// TIA Portal project "Esteira_3_V13_SP2_V14_V15" (V15)

(* hardware
DEVICE "S71500/ET200MP station_1"  S7-1500 station
   slot 0: "Rail_0"  6ES7 590-1***0-0AA0
   slot 1: "10D02_PLC"  CPU 1515F-2 PN  6ES7 515-2FM01-0AB0  V1.8
   slot 2: "F-DI 16x24V DC_1"  F-DI 16x24V DC  6ES7 526-1BH00-0AB0  V1.0
      slot 1: "F-DI 16x24V DC_1"  F-DI 16x24V DC  6ES7 526-1BH00-0AB0
   slot 3: "DI 16x24VDC BA_1"  DI 16x24VDC BA  6ES7 521-1BH10-0AA0  V1.0
   slot 4: "DQ 16x24VDC/0.5A BA_1"  DQ 16x24VDC/0.5A BA  6ES7 522-1BH10-0AA0  V1.0
DEVICE "25IHM01"  TP900 Comfort
   slot 0: "HMI"  HMI  6AV2 124-0JC01-0AX0  13.0.1.0
   slot 1: "HMI_RT_1"  TP900 Comfort  6AV2 124-0JC01-0AX0  13.0.1.0
   slot 5: "25IHM01.IE_CP_1"  PROFINET Interface
      slot 1: "PROFINET Interface_1"  PROFINET Interface
         slot 1: "Port_1"  Port
         slot 2: "Port_2"  Port
   slot 7: "25IHM01.MPI/DP_CP_1"  MPI/DP Interface
DEVICE "GSD device_4"  GSD.Device.PN
   slot 0: "Rack"  Rail  V1.0
   slot 0: "21U01_MVK-MPNIO-F"  55556
DEVICE "GSD device_5"  GSD.Device.PN
   slot 0: "Rack"  Rail  V1.0
   slot 0: "20U01_MVK-MPNIO-F"  55556
DEVICE "GSD device_6"  GSD.Device.PN
   slot 0: "Rack"  Rail  V1.0
   slot 0: "09U02_SEW-MDX61B-DFE32B"  182x xxx x  V1.4
      slot 0: "MDX61B+DFE32B V1.4"  182x xxx x  V1.4
DEVICE "SCALANCE X005"  SCALANCE X-Station
   slot 0: "SCALANCE X rack"  Rail
   slot 0: "Switch_1"  6GK5 005-0BA00-1AB2  V1.0
DEVICE "SCALANCE X005_1"  SCALANCE X-Station
   slot 0: "SCALANCE X rack"  Rail
   slot 0: "Switch_2"  6GK5 005-0BA00-1AB2  V1.0
DEVICE "GSD device_1"  GSD.Device.PN
   slot 0: "Rack"  Rail  V1.0
   slot 0: "19U02_Cube67-BN-PNIO"  56526  2
   slot 5: "21U05_56601 DIO16 E 8xM12_2"  56601
   slot 7: "20U05_56601 DIO16 E 8xM12_1"  56601
*)

// ===== PLC "10D02_PLC"  CPU 1515F-2 PN =====
// protected blocks, not shown: "Main_Safety_RTG1", "Main_Safety_RTG1_DB"

VAR_GLOBAL   // PLC tag table "Default tag table"
   "M_Estacao1_Andon" AT %M50.0 : Bool;
   "System_Byte" AT %MB1 : Byte;
   "FirstScan" AT %M1.0 : Bool;
   "DiagStatusUpdate" AT %M1.1 : Bool;
   "AlwaysTRUE" AT %M1.2 : Bool;
   "AlwaysFALSE" AT %M1.3 : Bool;
   "Clock_Byte" AT %MB0 : Byte;
   "Clock_10Hz" AT %M0.0 : Bool;
   "Clock_5Hz" AT %M0.1 : Bool;
   "Clock_2.5Hz" AT %M0.2 : Bool;
   "Clock_2Hz" AT %M0.3 : Bool;
   "Clock_1.25Hz" AT %M0.4 : Bool;
   "Clock_1Hz" AT %M0.5 : Bool;
   "Clock_0.625Hz" AT %M0.6 : Bool;
   "Clock_0.5Hz" AT %M0.7 : Bool;
   "Sempre_0" AT %M2.0 : Bool;
   "IHM_Tempo_Takt" AT %MD4 : Time;
   "IHM_Contagem_Tempo" AT %MD8 : Time;
   "11ME01_Emergência¶Painel Principal" AT %I0.0 : Bool;
   "11ME01_Reserva" AT %I0.1 : Bool;
   "11ME01_Reserva(1)" AT %I0.2 : Bool;
   "11ME01_Reserva(2)" AT %I0.3 : Bool;
   "11ME01_Reserva(3)" AT %I0.4 : Bool;
   "11ME01_Reserva(4)" AT %I0.5 : Bool;
   "11ME01_Reserva(5)" AT %I0.6 : Bool;
   "11ME01_Reserva(6)" AT %I0.7 : Bool;
   "11ME01_Emergência¶Painel Principal(1)" AT %I1.0 : Bool;
   "11ME01_Reserva(7)" AT %I1.1 : Bool;
   "11ME01_Reserva(8)" AT %I1.2 : Bool;
   "11ME01_Reset" AT %I1.3 : Bool;
   "11ME01_Reserva(9)" AT %I1.4 : Bool;
   "11ME01_Reserva(10)" AT %I1.5 : Bool;
   "11ME01_Reserva(11)" AT %I1.6 : Bool;
   "11ME01_Reserva(12)" AT %I1.7 : Bool;
   "12ME02_Termostato¶Painel" AT %I12.0 : Bool;
   "12ME02_Disjuntor¶Serviço Ok" AT %I12.1 : Bool;
   "12ME02_Disjuntor¶Tomada Ok" AT %I12.2 : Bool;
   "12ME02_Disjuntor¶Iluminação Ok" AT %I12.3 : Bool;
   "12ME02_Disjuntor¶Ar Condicionado Ok" AT %I12.4 : Bool;
   "12ME02_Disjuntor¶08F03 Ok" AT %I12.5 : Bool;
   "12ME02_Disjuntor¶Freio Ok" AT %I12.6 : Bool;
   "12ME02_Disjuntor¶Drive Ok" AT %I12.7 : Bool;
   "12ME02_Aquecimento¶Resistor Frenagem" AT %I13.0 : Bool;
   "12ME02_Disjuntor¶Ventilação Ok" AT %I13.1 : Bool;
   "12ME02_Reset_Emergencia" AT %I13.2 : Bool;
   "12ME02_Reserva(1)" AT %I13.3 : Bool;
   "12ME02_Reserva(2)" AT %I13.4 : Bool;
   "12ME02_Reserva(3)" AT %I13.5 : Bool;
   "12ME02_Reserva(4)" AT %I13.6 : Bool;
   "12ME02_Reserva(5)" AT %I13.7 : Bool;
   "15MS02_Reserva" AT %Q5.0 : Bool;
   "15MS02_Sirene_Giro" AT %Q5.1 : Bool;
   "15MS02_Reserva(2)" AT %Q5.2 : Bool;
   "15MS02_Reset" AT %Q5.3 : Bool;
   "15MS02_Torre de Sinalização¶Azul" AT %Q5.4 : Bool;
   "15MS02_Torre de Sinalização¶Verde" AT %Q5.5 : Bool;
   "15MS02_Torre de Sinalização¶Amarela" AT %Q5.6 : Bool;
   "15MS02_Torre de Sinalização¶Vermelha" AT %Q5.7 : Bool;
   "15MS02_Liga Ventilação¶Forçada" AT %Q6.0 : Bool;
   "15MS02_Reset_Rele_Emergencia" AT %Q6.1 : Bool;
   "15MS02_Reserva(4)" AT %Q6.2 : Bool;
   "15MS02_Reserva(5)" AT %Q6.3 : Bool;
   "15MS02_Reserva(6)" AT %Q6.4 : Bool;
   "15MS02_Reserva(7)" AT %Q6.5 : Bool;
   "15MS02_Reserva(8)" AT %Q6.6 : Bool;
   "15MS02_Reserva(9)" AT %Q6.7 : Bool;
   "20U1_Ack_Necessario" AT %I25.0 : Bool;
   "21U1_Ack_Necessario" AT %I34.0 : Bool;
   "22U1_Ack_Necessario" AT %I37.0 : Bool;
   "23U1_Ack_Necessario" AT %I68.0 : Bool;
   "20U1_GRUPO_OK" AT %I25.1 : Bool;
   "21U1_GRUPO_OK" AT %I34.1 : Bool;
   "22U1_GRUPO_OK" AT %I37.1 : Bool;
   "23U1_GRUPO_OK" AT %I68.1 : Bool;
   "IHM_Alarmes_Teste" AT %MB3 : Byte;
   "Contador_Cabinas" AT %MW12 : Int;
   "Ciclo_Giro" AT %MW14 : Word;
   "TESTES_MANUAIS" AT %M2.3 : Bool;
   "TESTE_LAMPADAS" AT %M20.0 : Bool;
END_VAR

VAR_GLOBAL   // PLC tag table "20U05"
   "20U05_Libera¶Estação 10" AT %I140.0 : Bool;
   "20U05_Reserva" AT %Q140.1 : Bool;
   "20U05_Libera¶Estação 20" AT %I140.2 : Bool;
   "20U05_Reserva(1)" AT %Q140.3 : Bool;
   "20U05_Reserva(2)" AT %I140.4 : Bool;
   "20U05_Reserva(3)" AT %Q140.5 : Bool;
   "20U05_Reserva(4)" AT %I140.6 : Bool;
   "20U05_Reserva(5)" AT %Q140.7 : Bool;
   "20U05_Apoio¶Estação 10" AT %I141.0 : Bool;
   "20U05_Reserva(6)" AT %Q141.1 : Bool;
   "20U05_Apoio¶Estação 20" AT %I141.2 : Bool;
   "20U05_Reserva(7)" AT %Q141.3 : Bool;
   "20U05_Reserva(8)" AT %I141.4 : Bool;
   "20U05_Reserva(9)" AT %Q141.5 : Bool;
   "20U05_Reserva(10)" AT %I141.6 : Bool;
   "20U05_Reserva(11)" AT %Q141.7 : Bool;
END_VAR

VAR_GLOBAL   // PLC tag table "20U01"
   "20U01_Reserva" AT %I116.0 : Bool;
   "20U01_Reserva(1)" AT %I116.1 : Bool;
   "20U01_Reserva(2)" AT %I116.2 : Bool;
   "20U01_Emergência¶Estação 1" AT %I116.3 : Bool;
   "20U01_Reserva(3)" AT %I116.4 : Bool;
   "20U01_Reserva(4)" AT %I116.5 : Bool;
   "20U01_Reserva(5)" AT %I116.6 : Bool;
   "20U01_Reserva(6)" AT %I116.7 : Bool;
   "20U01_Emergência¶Estação 2" AT %I117.0 : Bool;
   "20U01_Reserva(7)" AT %I117.1 : Bool;
   "20U01_Reserva(8)" AT %I117.2 : Bool;
   "20U01_Reserva(9)" AT %I117.3 : Bool;
   "20U01_Reserva(10)" AT %I117.4 : Bool;
   "20U01_Reserva(11)" AT %I117.5 : Bool;
   "20U01_Reserva(12)" AT %I117.6 : Bool;
   "20U01_Reserva(13)" AT %I117.7 : Bool;
   "20U1_Reseta_Modulo" AT %Q7.0 : Bool;
   "Muting_Cortina" AT %M2.1 : Bool;
   "Emergencia_Cortina" AT %M2.2 : Bool;
END_VAR

VAR_GLOBAL   // PLC tag table "21U01"
   "21U01_Cortina_Saida" AT %I122.0 : Bool;
   "21U01_Reserva(1)" AT %I122.1 : Bool;
   "21U01_Reserva(2)" AT %I122.2 : Bool;
   "21U01_Emergência¶Estação 3" AT %I122.3 : Bool;
   "21U01_Reserva(3)" AT %I122.4 : Bool;
   "21U01_Reserva(4)" AT %I122.5 : Bool;
   "21U01_Reserva(5)" AT %I122.6 : Bool;
   "21U01_Reserva(6)" AT %I122.7 : Bool;
   "21U01_Emergência¶Estação 4" AT %I123.0 : Bool;
   "21U01_Reserva(7)" AT %I123.1 : Bool;
   "21U01_Reserva(8)" AT %I123.2 : Bool;
   "21U01_Reserva(9)" AT %I123.3 : Bool;
   "21U01_Reserva(10)" AT %I123.4 : Bool;
   "21U01_Reserva(11)" AT %I123.5 : Bool;
   "21U01_Reserva(12)" AT %I123.6 : Bool;
   "21U01_Reserva(13)" AT %I123.7 : Bool;
   "21U1_Reseta_Modulo" AT %Q8.0 : Bool;
END_VAR

VAR_GLOBAL   // PLC tag table "21U05"
   "21U05_Libera¶Estação 30" AT %I144.0 : Bool;
   "21U05_Reserva" AT %Q144.1 : Bool;
   "21U05_Libera¶Estação 40" AT %I144.2 : Bool;
   "21U05_Reserva(1)" AT %Q144.3 : Bool;
   "21U05_Cabine_Retirada" AT %I144.4 : Bool;
   "21U05_Reserva(3)" AT %Q144.5 : Bool;
   "21U05_Reserva(4)" AT %I144.6 : Bool;
   "21U05_Reserva(5)" AT %Q144.7 : Bool;
   "21U05_Apoio¶Estação 30" AT %I145.0 : Bool;
   "21U05_Reserva(6)" AT %Q145.1 : Bool;
   "21U05_Apoio¶Estação 40" AT %I145.2 : Bool;
   "21U05_Reserva(7)" AT %Q145.3 : Bool;
   "21U05_Reserva(8)" AT %I145.4 : Bool;
   "21U05_Reserva(9)" AT %Q145.5 : Bool;
   "21U05_Reserva(10)" AT %I145.6 : Bool;
   "21U05_Reserva(11)" AT %Q145.7 : Bool;
END_VAR

DATA_BLOCK "ANDON_DB"   // DB2
{ S7_Optimized_Access := 'TRUE' }
VERSION : 0.1
// stored: InstanceOfName ANDON
"ANDON"
BEGIN
END_DATA_BLOCK

DATA_BLOCK "Multiplo_Uso_DB"   // DB5
{ S7_Optimized_Access := 'TRUE' }
VERSION : 0.1
   VAR
      HORA_Atual : Time_Of_Day;
      DATA_Atual : DTL;
   END_VAR
   VAR RETAIN
      T_Takt : IEC_COUNTER;
   END_VAR
   VAR
      retorno_Data : Int;
   END_VAR
   VAR RETAIN
      INICIO_JORNADA : DTL;
      FINAL_JORNADA : DTL;
      INICIO_ALMOÇO : DTL;
   END_VAR
   VAR
      FINAL_ALMOÇO : DTL;
      EM_JORNADA : Bool;
      EM_JORNADA_CMP : Bool;
   END_VAR
   VAR RETAIN
      IHM_TAKT_MINUTOS : Int;
      IHM_TAKT_SEGUNDOS : Int;
      TAKT_SEGUNDOS : Int;
   END_VAR
   VAR
      FINAL_DO_TAKT : Bool;
      Contagem_Takt : Int;
      Emergencia_Principal_OK : Bool;
      Emergencia_OP10_OK : Bool;
      Emergencia_OP20_OK : Bool;
      Emergencia_OP30_OK : Bool;
      Emergencia_OP40_OK : Bool;
      Emergencia_OP50_OK : Bool;
      Emergencia_OP60_OK : Bool;
      Emergencia_OP70_OK : Bool;
      Emergencia_OP80_OK : Bool;
      EMERGENCIAS_OK : Bool;
      OPERACAO10_OK : Bool;
      OPERACAO20_OK : Bool;
      OPERACAO30_OK : Bool;
      OPERACAO40_OK : Bool;
      OPERACAO50_OK : Bool;
      OPERACAO60_OK : Bool;
      OPERACAO70_OK : Bool;
      OPERACAO80_OK : Bool;
      OPERACOES_OK : Bool;
      Roda_Linha : Bool;
      Roda_Linha_cmp : Bool;
   END_VAR
   VAR RETAIN
      CONTAGEM_CABINAS : Int;
      TOTAL_CABINAS_TURNO : Int;
   END_VAR
   VAR
      GMT_Brasilia : Time := T#3h;
      Fim_De_Producao : Bool;
      Fim_De_Producao_cmp : Bool;
   END_VAR
   VAR RETAIN
      DESABILITA_OP10 : Bool;
      DESABILITA_OP20 : Bool;
      DESABILITA_OP30 : Bool;
      DESABILITA_OP40 : Bool;
      DESABILITA_OP50 : Bool;
      DESABILITA_OP60 : Bool;
      DESABILITA_OP70 : Bool;
      DESABILITA_OP80 : Bool;
      IHM_Velocidade_Automatico : Int := 10;
      IHM_Velocidade_Manual : Int := 4;
      IHM_Descolamento_Cabinas_mm : DInt := 5825;
   END_VAR
   VAR
      IHM_Modo_Manual : Bool;
      IHM_Modo_Manual_cmp : Bool;
      IHM_Modo_Automatico : Bool;
      IHM_Modo_Automatico_cmp : Bool;
      IHM_Jog_CW : Bool;
      IHM_Jog_CCW : Bool;
      IHM_Posicao_Atual : DInt;
      IHM_Velocidade_Atual : Int;
      T_RESET_RELE_SEG : IEC_TIMER;
      IHM_HABILITA_DRIVER : Bool;
      IHM_HABILITA_DRIVER_CMP : Bool;
      ZERA_POSICAO : Bool;
      RESETA_TAKT : Bool;
      PARAR_OP10 : Bool;
      PARAR_OP20 : Bool;
      PARAR_OP30 : Bool;
      PARAR_OP40 : Bool;
      PARAR_OP50 : Bool;
      PARAR_OP60 : Bool;
      PARAR_OP70 : Bool;
      PARAR_OP80 : Bool;
      Ciclo_Giro : Int;
      Shifter_Giro : Bool;
      T_Reset_Takt : IEC_TIMER;
      T_Retirada_Cabine : IEC_TIMER;
      CABINE_RETIRADA : Bool;
      Emergencia_Cortina_Saida_OK : Bool;
      Muting_Cortina : Bool;
      T_SIRENE : IEC_TIMER;
      Sirene_Giro : Bool;
      Tempo_Sirene : Time;
   END_VAR
   VAR RETAIN
      IHM_Tempo_Aviso1 : Int;
      IHM_Tempo_Aviso2 : Int;
   END_VAR
   VAR
      Inicio_Aviso1 : Int;
      Final_Aviso1 : Int;
      Inicio_Aviso2 : Int;
      Final_Aviso2 : Int;
      IHM_Zerar_Contagem : Bool;
      IHM_Zerar_Posicao_Esteira : Bool;
      IHM_Zerar_Takt : Bool;
      Tempo_OP10 : Int;
      Tempo_OP20 : Int;
      Tempo_OP30 : Int;
      Tempo_OP40 : Int;
      Stop_Time_OP10 : Int;
      Stop_Time_OP20 : Int;
      Stop_Time_OP30 : Int;
      Stop_Time_OP40 : Int;
   END_VAR
BEGIN
END_DATA_BLOCK

DATA_BLOCK "ALARMES_DB"   // DB12
{ S7_Optimized_Access := 'FALSE' }
VERSION : 0.1
   VAR
      DBW0 : Int;
      DBW1 : Int;
      DBW2 : Int;
      DBW3 : Int;
   END_VAR
BEGIN
END_DATA_BLOCK

DATA_BLOCK "DB_Global_Sistema"   // DB23
{ S7_Optimized_Access := 'FALSE' }
VERSION : 0.1
   VAR
      TEMPO_TAKT : Int;
      Apoio_OP10 : Bool;
      Apoio_OP20 : Bool;
      Apoio_OP30 : Bool;
      Apoio_OP40 : Bool;
      Apoio_OP50 : Bool;
      Apoio_OP60 : Bool;
      Apoio_OP70 : Bool;
      Apoio_OP80 : Bool;
      Contagem_Cabinas : Int;
      Stop_Time : Int;
      Cabinas_Programadas : Int;
   END_VAR
BEGIN
END_DATA_BLOCK

DATA_BLOCK "Modulo_259"   // DB286
{ S7_Optimized_Access := 'TRUE' }
VERSION : 0.1
   VAR
      IO_ADDRESS_or_HW_IDENTIFIER : Hw_Io := 318;   // S71xxxx: assign HW_Identifier; S74xx/3xx assign Peripheral address
      INHIBIT : Bool;   // false: Contr. inhibit; true: enable
      ENABLE_RAPID_STOP : Bool;   // false: rapid stop; true: enable
      ENABLE : Bool;   // false: stop; true: enable
      RESET : Bool;
      Start : Bool;
      JOG_PLUS_MODE : Bool;   // select Jog+_Mode
      JOG_MINUS_MODE : Bool;   // select Jog-_Mode
      REF_TRAVEL_MODE : Bool;   // select Reference_Travel_Mode
      AUTO_OPT : Bool;   // select AUTO_OPT_Mode
      AUTO_CW : Bool;   // select AUTO_CW_Mode
      AUTO_CCW : Bool;   // select AUTO_CCW_Mode
      AUTO_PULS_CW : Bool;   // select AUTO_PULS_CW_Mode
      AUTO_PULS_CCW : Bool;   // select AUTO_PULS_CCW_Mode
      SETPOINT_POS : DInt := 0;
      SETPOINT_SPEED : Int := 4;
      START_RAMP : Int := 1001;   // Attention: Avoid Ramp = 0!
      STOP_RAMP : Int := 2002;   // Attention: Avoid Ramp = 0!
      COMMUNICATION_OK : Bool;   // DPRD_DAT & DPWR_DAT: Return Value = 0 / SFC14/SFC15: Return Value = 0
      FAULT_OF_AXIS : Bool;   // A fault is active, if the inverter is not ready for operation AND the error bit has been set.
      WARNING_OF_AXIS : Bool;   // A warning is active, if the inverter is still ready for operation AND the error bit has been set.
      INVERTER_READY : Bool;
      REFERENCED : Bool;
      TARGET_POS_REACHED : Bool;
      AXIS_INTERLOCKED : Bool;   // mode selection is illogical (no mode or several modes selected) / die Modeanwahl ist unplausibel (kein Mode oder mehrere Modi angewählt)
      FAULT_NO : Int;
      ACTUAL_POSITION : DInt;
      ACTUAL_SPEED : Int;
      ACTUAL_CURRENT : Int;
   END_VAR
BEGIN
END_DATA_BLOCK

// folder: BANCO

DATA_BLOCK "Banco_Hora_Operacoes"   // DB13
{ S7_Optimized_Access := 'FALSE' }
VERSION : 0.1
   VAR
      Produto_1 : Struct
         Data_e_Hora : DTL;
         Tempo_OP10 : Int;
         Tempo_OP20 : Int;
         Tempo_OP30 : Int;
         Tempo_OP40 : Int;
         Tempo_OP50 : Int;
         Tempo_OP60 : Int;
         Tempo_OP70 : Int;
         Tempo_OP80 : Int;
         Stop_Time_OP10 : Int;
         Stop_Time_OP20 : Int;
         Stop_Time_OP30 : Int;
         Stop_Time_OP40 : Int;
         Stop_Time_OP50 : Int;
         Stop_Time_OP60 : Int;
         Stop_Time_OP70 : Int;
         Stop_Time_OP80 : Int;
      END_STRUCT;
   END_VAR
BEGIN
END_DATA_BLOCK

// folder: DB_OPERACOES

DATA_BLOCK "Operacao_20_DB"   // DB3
{ S7_Optimized_Access := 'TRUE' }
VERSION : 0.1
// stored: InstanceOfName Operacao
"Operacao"
BEGIN
END_DATA_BLOCK

DATA_BLOCK "Operacao_10_DB"   // DB4
{ S7_Optimized_Access := 'TRUE' }
VERSION : 0.1
// stored: InstanceOfName Operacao
"Operacao"
BEGIN
END_DATA_BLOCK

DATA_BLOCK "Operacao_30_DB"   // DB6
{ S7_Optimized_Access := 'TRUE' }
VERSION : 0.1
// stored: InstanceOfName Operacao
"Operacao"
BEGIN
END_DATA_BLOCK

DATA_BLOCK "Operacao_40_DB"   // DB7
{ S7_Optimized_Access := 'TRUE' }
VERSION : 0.1
// stored: InstanceOfName Operacao
"Operacao"
BEGIN
END_DATA_BLOCK

DATA_BLOCK "Operacao_50_DB"   // DB8
{ S7_Optimized_Access := 'TRUE' }
VERSION : 0.1
// stored: InstanceOfName Operacao
"Operacao"
BEGIN
END_DATA_BLOCK

DATA_BLOCK "Operacao_60_DB"   // DB9
{ S7_Optimized_Access := 'TRUE' }
VERSION : 0.1
// stored: InstanceOfName Operacao
"Operacao"
BEGIN
END_DATA_BLOCK

DATA_BLOCK "Operacao_70_DB"   // DB10
{ S7_Optimized_Access := 'TRUE' }
VERSION : 0.1
// stored: InstanceOfName Operacao
"Operacao"
BEGIN
END_DATA_BLOCK

DATA_BLOCK "Operacao_80_DB"   // DB11
{ S7_Optimized_Access := 'TRUE' }
VERSION : 0.1
// stored: InstanceOfName Operacao
"Operacao"
BEGIN
END_DATA_BLOCK

// folder: (top level)

FUNCTION_BLOCK "Operacao"   // FB2, LAD
{ S7_Optimized_Access := 'TRUE' }
VERSION : 0.1
   VAR_INPUT
      Parar_Linha : Bool;
      Emergencia_OK : Bool;
      Emergencia_OP_OK : Bool;
   END_VAR
   VAR_OUTPUT
      Operacao_OK : Bool;
      Tempo_Da_Operacao : Int;
      Stop_Time : Int;
   END_VAR
   VAR
      Operacao_OK_cmp : Bool;
   END_VAR
   VAR_TEMP   // added for the SCL form of the ladder/FBD networks
      _w1 : Bool;
   END_VAR
BEGIN

REGION Network 1: operacao ok
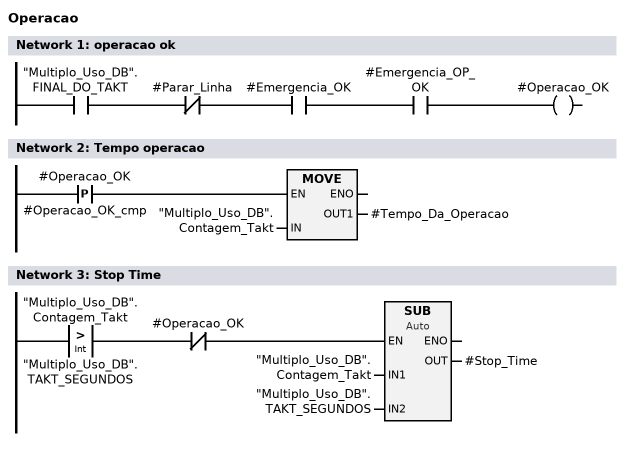
   RUNG wire#powerrail
      Contact( "Multiplo_Uso_DB".FINAL_DO_TAKT )
      I_Contact( #Parar_Linha )
      Contact( #Emergencia_OK )
      Contact( #Emergencia_OP_OK )
      Coil( #Operacao_OK )
   END_RUNG
   // the same network as SCL:
   #Operacao_OK := "Multiplo_Uso_DB".FINAL_DO_TAKT AND NOT #Parar_Linha AND #Emergencia_OK AND #Emergencia_OP_OK;
END_REGION

REGION Network 2: Tempo operacao
   RUNG wire#powerrail
      P_Contact(operand := #Operacao_OK, bit := #Operacao_OK_cmp)
      Move(in := "Multiplo_Uso_DB".Contagem_Takt, out1 => #Tempo_Da_Operacao)
   END_RUNG
   // the same network as SCL:
   #_w1 := #Operacao_OK AND NOT #Operacao_OK_cmp;   // rising edge of #Operacao_OK
   #Operacao_OK_cmp := #Operacao_OK;
   IF #_w1 THEN #Tempo_Da_Operacao := "Multiplo_Uso_DB".Contagem_Takt; END_IF;
END_REGION

REGION Network 3: Stop Time
   RUNG wire#powerrail
      { S7_Templates := "SrcType := Int" } GT_Contact(in1 := "Multiplo_Uso_DB".Contagem_Takt, in2 := "Multiplo_Uso_DB".TAKT_SEGUNDOS)
      I_Contact( #Operacao_OK )
      Sub(in1 := "Multiplo_Uso_DB".Contagem_Takt, in2 := "Multiplo_Uso_DB".TAKT_SEGUNDOS, out => #Stop_Time)
   END_RUNG
   // the same network as SCL:
   IF ("Multiplo_Uso_DB".Contagem_Takt > "Multiplo_Uso_DB".TAKT_SEGUNDOS) AND NOT #Operacao_OK THEN
       #Stop_Time := "Multiplo_Uso_DB".Contagem_Takt - "Multiplo_Uso_DB".TAKT_SEGUNDOS;
   END_IF;
END_REGION
END_FUNCTION_BLOCK

FUNCTION_BLOCK "ANDON"   // FB3, LAD
{ S7_Optimized_Access := 'TRUE' }
VERSION : 0.1
   VAR_INPUT
      FINAL_JORNADA : DTL;
      INICIO_JORNADA : DTL;
      INICIO_ALMOÇO : DTL;
   END_VAR
   VAR_OUTPUT
      EM_JORNADA : Bool;
      FINAL_DE_TAKT : Bool;
   END_VAR
   VAR
      FINAL_ALMOÇO : DTL;
      INICIAR_CONTAGEM : Bool;
      INICIAR_CONTAGEM_cmp : Bool;
      MINUTOS_P_SEGUNDOS : Int;
      T_SIRENE_INT : Int;
   END_VAR
BEGIN

REGION Network 1
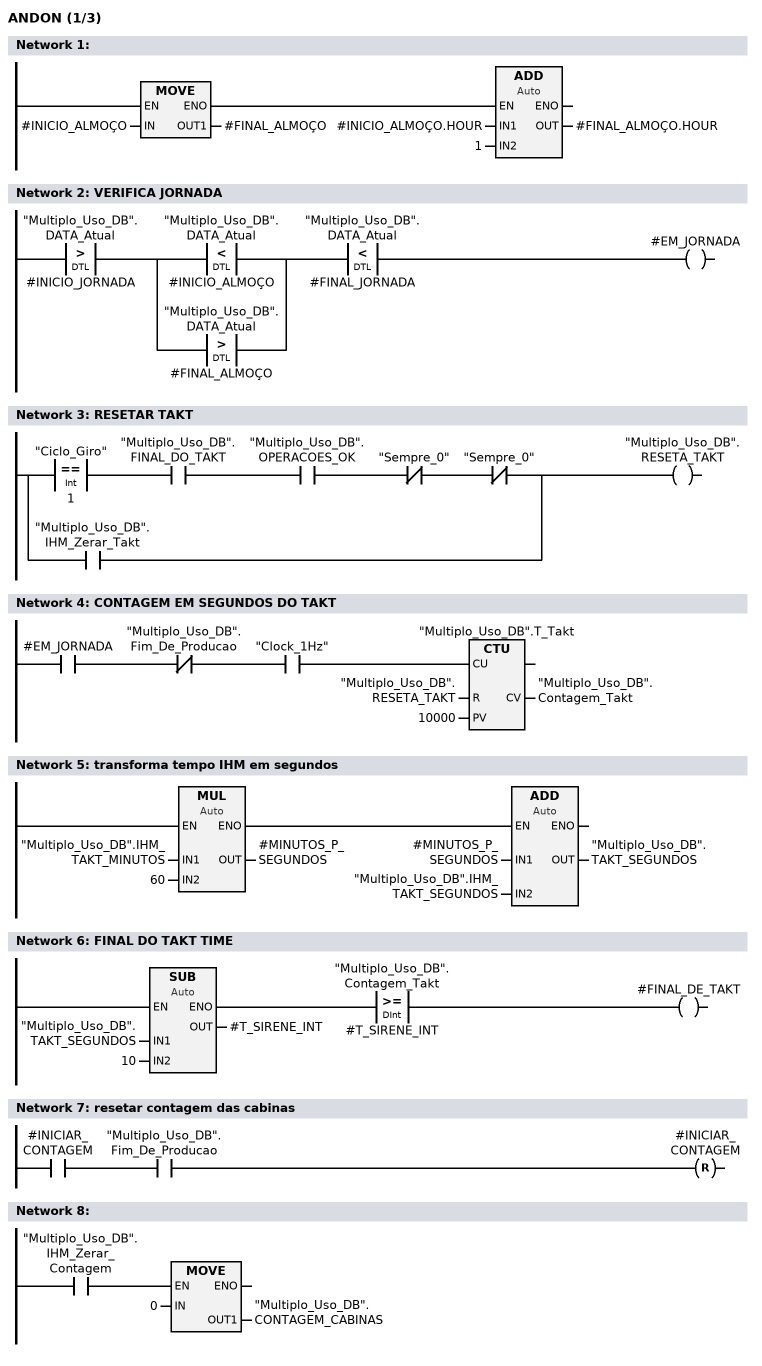
   RUNG wire#powerrail
      Move(in := #INICIO_ALMOÇO, out1 => #FINAL_ALMOÇO)
      Add(in1 := #INICIO_ALMOÇO.HOUR, in2 := 1, out => #FINAL_ALMOÇO.HOUR)
   END_RUNG
   // the same network as SCL:
   #FINAL_ALMOÇO := #INICIO_ALMOÇO;
   #FINAL_ALMOÇO.HOUR := #INICIO_ALMOÇO.HOUR + 1;
END_REGION

REGION Network 2: VERIFICA JORNADA
   RUNG wire#powerrail
      { S7_Templates := "SrcType := DTL" } GT_Contact(in1 := "Multiplo_Uso_DB".DATA_Atual, in2 := #INICIO_JORNADA)
      wire#w1
      { S7_Templates := "SrcType := DTL" } LT_Contact(in1 := "Multiplo_Uso_DB".DATA_Atual, in2 := #INICIO_ALMOÇO)
      wire#w2
      { S7_Templates := "SrcType := DTL" } LT_Contact(in1 := "Multiplo_Uso_DB".DATA_Atual, in2 := #FINAL_JORNADA)
      Coil( #EM_JORNADA )
   END_RUNG
   RUNG wire#w1
      { S7_Templates := "SrcType := DTL" } GT_Contact(in1 := "Multiplo_Uso_DB".DATA_Atual, in2 := #FINAL_ALMOÇO)
   END_RUNG wire#w2
   // the same network as SCL:
   #EM_JORNADA := ("Multiplo_Uso_DB".DATA_Atual > #INICIO_JORNADA) AND (("Multiplo_Uso_DB".DATA_Atual < #INICIO_ALMOÇO) OR ("Multiplo_Uso_DB".DATA_Atual > #FINAL_ALMOÇO)) AND ("Multiplo_Uso_DB".DATA_Atual < #FINAL_JORNADA);
END_REGION

REGION Network 3: RESETAR TAKT
   RUNG wire#powerrail
      { S7_Templates := "SrcType := Int" } EQ_Contact(in1 := "Ciclo_Giro", in2 := 1)
      Contact( "Multiplo_Uso_DB".FINAL_DO_TAKT )
      Contact( "Multiplo_Uso_DB".OPERACOES_OK )
      I_Contact( "Sempre_0" )
      I_Contact( "Sempre_0" )
      wire#w1
      Coil( "Multiplo_Uso_DB".RESETA_TAKT )
   END_RUNG
   RUNG wire#powerrail
      Contact( "Multiplo_Uso_DB".IHM_Zerar_Takt )
   END_RUNG wire#w1
   // the same network as SCL:
   "Multiplo_Uso_DB".RESETA_TAKT := (("Ciclo_Giro" = 1) AND "Multiplo_Uso_DB".FINAL_DO_TAKT AND "Multiplo_Uso_DB".OPERACOES_OK AND NOT "Sempre_0" AND NOT "Sempre_0") OR "Multiplo_Uso_DB".IHM_Zerar_Takt;
END_REGION

REGION Network 4: CONTAGEM EM SEGUNDOS DO TAKT
   "Multiplo_Uso_DB".T_Takt.CTU(CU := #EM_JORNADA AND NOT "Multiplo_Uso_DB".Fim_De_Producao AND "Clock_1Hz",
                           R := "Multiplo_Uso_DB".RESETA_TAKT,
                           PV := 10000,
                           CV => "Multiplo_Uso_DB".Contagem_Takt);
END_REGION

REGION Network 5: transforma tempo IHM em segundos
   RUNG wire#powerrail
      Mul(in1 := "Multiplo_Uso_DB".IHM_TAKT_MINUTOS, in2 := 60, out => #MINUTOS_P_SEGUNDOS)
      Add(in1 := #MINUTOS_P_SEGUNDOS, in2 := "Multiplo_Uso_DB".IHM_TAKT_SEGUNDOS, out => "Multiplo_Uso_DB".TAKT_SEGUNDOS)
   END_RUNG
   // the same network as SCL:
   #MINUTOS_P_SEGUNDOS := "Multiplo_Uso_DB".IHM_TAKT_MINUTOS * 60;
   "Multiplo_Uso_DB".TAKT_SEGUNDOS := #MINUTOS_P_SEGUNDOS + "Multiplo_Uso_DB".IHM_TAKT_SEGUNDOS;
END_REGION

REGION Network 6: FINAL DO TAKT TIME
   RUNG wire#powerrail
      Sub(in1 := "Multiplo_Uso_DB".TAKT_SEGUNDOS, in2 := 10, out => #T_SIRENE_INT)
      { S7_Templates := "SrcType := DInt" } GE_Contact(in1 := "Multiplo_Uso_DB".Contagem_Takt, in2 := #T_SIRENE_INT)
      Coil( #FINAL_DE_TAKT )
   END_RUNG
   // the same network as SCL:
   #T_SIRENE_INT := "Multiplo_Uso_DB".TAKT_SEGUNDOS - 10;
   #FINAL_DE_TAKT := "Multiplo_Uso_DB".Contagem_Takt >= #T_SIRENE_INT;
END_REGION

REGION Network 7: resetar contagem das cabinas
   RUNG wire#powerrail
      Contact( #INICIAR_CONTAGEM )
      Contact( "Multiplo_Uso_DB".Fim_De_Producao )
      R_Coil( #INICIAR_CONTAGEM )
   END_RUNG
   // the same network as SCL:
   IF #INICIAR_CONTAGEM AND "Multiplo_Uso_DB".Fim_De_Producao THEN #INICIAR_CONTAGEM := FALSE; END_IF;
END_REGION

REGION Network 8
   RUNG wire#powerrail
      Contact( "Multiplo_Uso_DB".IHM_Zerar_Contagem )
      Move(in := 0, out1 => "Multiplo_Uso_DB".CONTAGEM_CABINAS)
   END_RUNG
   // the same network as SCL:
   IF "Multiplo_Uso_DB".IHM_Zerar_Contagem THEN "Multiplo_Uso_DB".CONTAGEM_CABINAS := 0; END_IF;
END_REGION

REGION Network 9: Sinaliza fim de produção
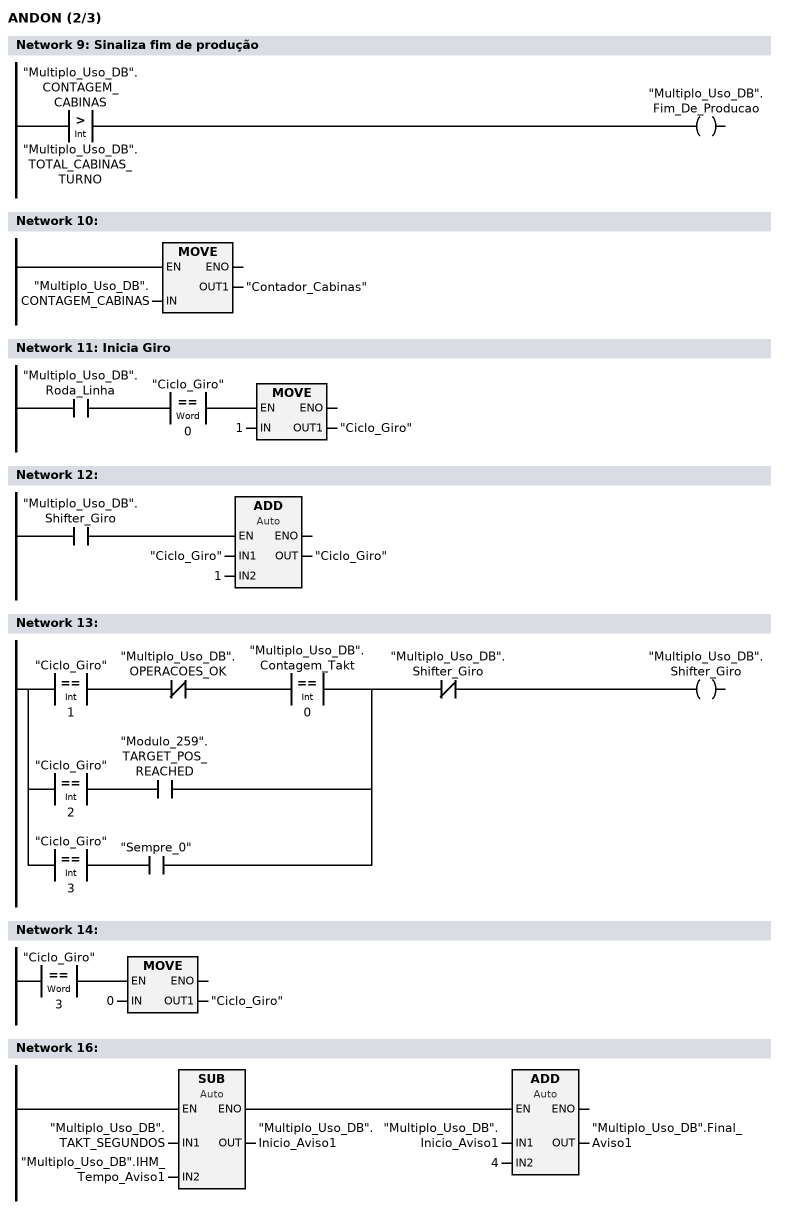
   RUNG wire#powerrail
      { S7_Templates := "SrcType := Int" } GT_Contact(in1 := "Multiplo_Uso_DB".CONTAGEM_CABINAS, in2 := "Multiplo_Uso_DB".TOTAL_CABINAS_TURNO)
      Coil( "Multiplo_Uso_DB".Fim_De_Producao )
   END_RUNG
   // the same network as SCL:
   "Multiplo_Uso_DB".Fim_De_Producao := "Multiplo_Uso_DB".CONTAGEM_CABINAS > "Multiplo_Uso_DB".TOTAL_CABINAS_TURNO;
END_REGION

REGION Network 10
   RUNG wire#powerrail
      Move(in := "Multiplo_Uso_DB".CONTAGEM_CABINAS, out1 => "Contador_Cabinas")
   END_RUNG
   // the same network as SCL:
   "Contador_Cabinas" := "Multiplo_Uso_DB".CONTAGEM_CABINAS;
END_REGION

REGION Network 11: Inicia Giro
   RUNG wire#powerrail
      Contact( "Multiplo_Uso_DB".Roda_Linha )
      { S7_Templates := "SrcType := Word" } EQ_Contact(in1 := "Ciclo_Giro", in2 := 0)
      Move(in := 1, out1 => "Ciclo_Giro")
   END_RUNG
   // the same network as SCL:
   IF "Multiplo_Uso_DB".Roda_Linha AND ("Ciclo_Giro" = 0) THEN "Ciclo_Giro" := 1; END_IF;
END_REGION

REGION Network 12
   RUNG wire#powerrail
      Contact( "Multiplo_Uso_DB".Shifter_Giro )
      Add(in1 := "Ciclo_Giro", in2 := 1, out => "Ciclo_Giro")
   END_RUNG
   // the same network as SCL:
   IF "Multiplo_Uso_DB".Shifter_Giro THEN "Ciclo_Giro" := "Ciclo_Giro" + 1; END_IF;
END_REGION

REGION Network 13
   RUNG wire#powerrail
      { S7_Templates := "SrcType := Int" } EQ_Contact(in1 := "Ciclo_Giro", in2 := 1)
      I_Contact( "Multiplo_Uso_DB".OPERACOES_OK )
      { S7_Templates := "SrcType := Int" } EQ_Contact(in1 := "Multiplo_Uso_DB".Contagem_Takt, in2 := 0)
      wire#w1
      I_Contact( "Multiplo_Uso_DB".Shifter_Giro )
      Coil( "Multiplo_Uso_DB".Shifter_Giro )
   END_RUNG
   RUNG wire#powerrail
      { S7_Templates := "SrcType := Int" } EQ_Contact(in1 := "Ciclo_Giro", in2 := 2)
      Contact( "Modulo_259".TARGET_POS_REACHED )
   END_RUNG wire#w1
   RUNG wire#powerrail
      { S7_Templates := "SrcType := Int" } EQ_Contact(in1 := "Ciclo_Giro", in2 := 3)
      Contact( "Sempre_0" )
   END_RUNG wire#w1
   // the same network as SCL:
   "Multiplo_Uso_DB".Shifter_Giro := ((("Ciclo_Giro" = 1) AND NOT "Multiplo_Uso_DB".OPERACOES_OK AND ("Multiplo_Uso_DB".Contagem_Takt = 0)) OR (("Ciclo_Giro" = 2) AND "Modulo_259".TARGET_POS_REACHED) OR (("Ciclo_Giro" = 3) AND "Sempre_0")) AND NOT "Multiplo_Uso_DB".Shifter_Giro;
END_REGION

REGION Network 14
   RUNG wire#powerrail
      { S7_Templates := "SrcType := Word" } EQ_Contact(in1 := "Ciclo_Giro", in2 := 3)
      Move(in := 0, out1 => "Ciclo_Giro")
   END_RUNG
   // the same network as SCL:
   IF "Ciclo_Giro" = 3 THEN "Ciclo_Giro" := 0; END_IF;
END_REGION

REGION Network 16
   RUNG wire#powerrail
      Sub(in1 := "Multiplo_Uso_DB".TAKT_SEGUNDOS, in2 := "Multiplo_Uso_DB".IHM_Tempo_Aviso1, out => "Multiplo_Uso_DB".Inicio_Aviso1)
      Add(in1 := "Multiplo_Uso_DB".Inicio_Aviso1, in2 := 4, out => "Multiplo_Uso_DB".Final_Aviso1)
   END_RUNG
   // the same network as SCL:
   "Multiplo_Uso_DB".Inicio_Aviso1 := "Multiplo_Uso_DB".TAKT_SEGUNDOS - "Multiplo_Uso_DB".IHM_Tempo_Aviso1;
   "Multiplo_Uso_DB".Final_Aviso1 := "Multiplo_Uso_DB".Inicio_Aviso1 + 4;
END_REGION

REGION Network 17
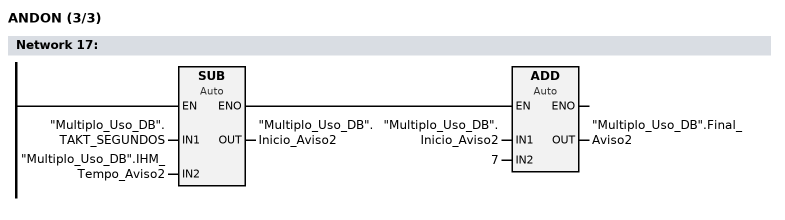
   RUNG wire#powerrail
      Sub(in1 := "Multiplo_Uso_DB".TAKT_SEGUNDOS, in2 := "Multiplo_Uso_DB".IHM_Tempo_Aviso2, out => "Multiplo_Uso_DB".Inicio_Aviso2)
      Add(in1 := "Multiplo_Uso_DB".Inicio_Aviso2, in2 := 7, out => "Multiplo_Uso_DB".Final_Aviso2)
   END_RUNG
   // the same network as SCL:
   "Multiplo_Uso_DB".Inicio_Aviso2 := "Multiplo_Uso_DB".TAKT_SEGUNDOS - "Multiplo_Uso_DB".IHM_Tempo_Aviso2;
   "Multiplo_Uso_DB".Final_Aviso2 := "Multiplo_Uso_DB".Inicio_Aviso2 + 7;
END_REGION
END_FUNCTION_BLOCK

FUNCTION "Reset_Rede" : Void   // FC1, LAD
{ S7_Optimized_Access := 'TRUE' }
VERSION : 0.1
BEGIN

REGION Network 1
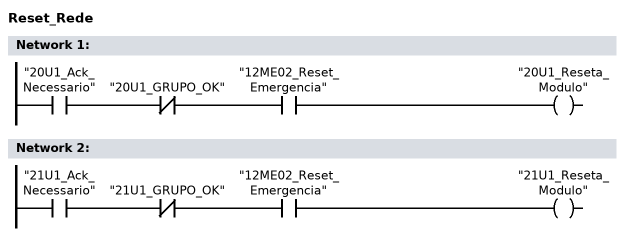
   RUNG wire#powerrail
      Contact( "20U1_Ack_Necessario" )
      I_Contact( "20U1_GRUPO_OK" )
      Contact( "12ME02_Reset_Emergencia" )
      Coil( "20U1_Reseta_Modulo" )
   END_RUNG
   // the same network as SCL:
   "20U1_Reseta_Modulo" := "20U1_Ack_Necessario" AND NOT "20U1_GRUPO_OK" AND "12ME02_Reset_Emergencia";
END_REGION

REGION Network 2
   RUNG wire#powerrail
      Contact( "21U1_Ack_Necessario" )
      I_Contact( "21U1_GRUPO_OK" )
      Contact( "12ME02_Reset_Emergencia" )
      Coil( "21U1_Reseta_Modulo" )
   END_RUNG
   // the same network as SCL:
   "21U1_Reseta_Modulo" := "21U1_Ack_Necessario" AND NOT "21U1_GRUPO_OK" AND "12ME02_Reset_Emergencia";
END_REGION
END_FUNCTION

FUNCTION "ALARMES" : Void   // FC2, LAD
{ S7_Optimized_Access := 'TRUE' }
VERSION : 0.1
BEGIN

REGION Network 1
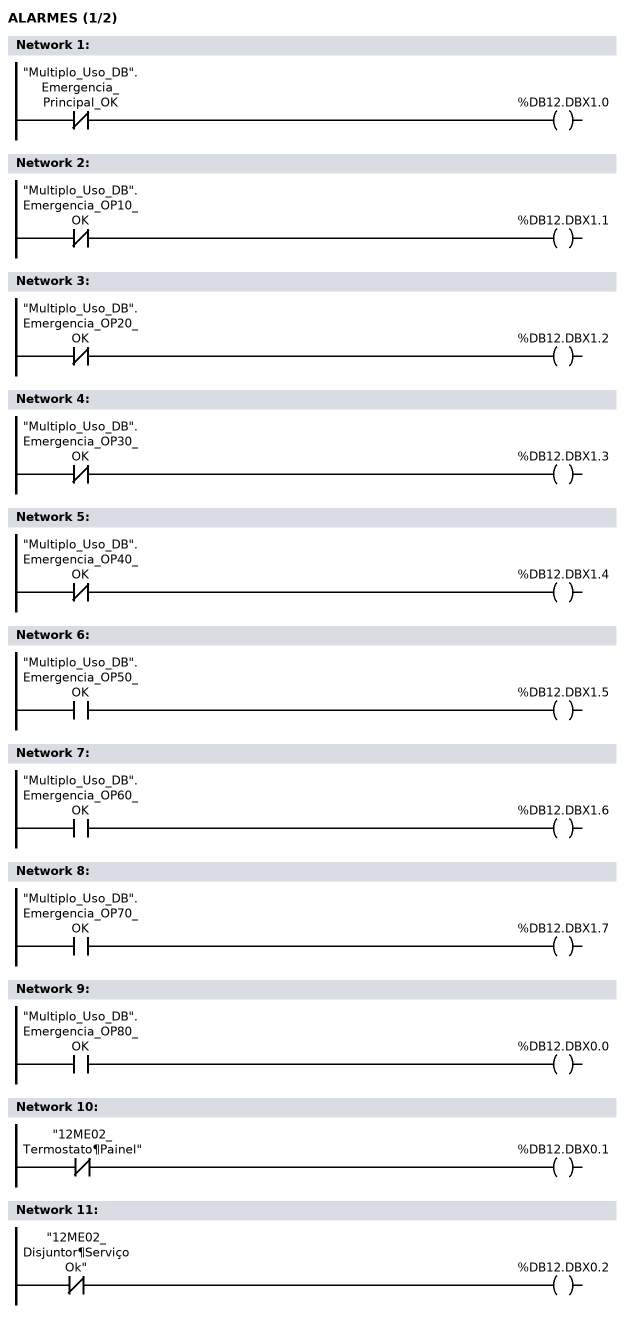
   RUNG wire#powerrail
      I_Contact( "Multiplo_Uso_DB".Emergencia_Principal_OK )
      Coil( %DB12.DBX1.0 )
   END_RUNG
   // the same network as SCL:
   %DB12.DBX1.0 := NOT "Multiplo_Uso_DB".Emergencia_Principal_OK;
END_REGION

REGION Network 2
   RUNG wire#powerrail
      I_Contact( "Multiplo_Uso_DB".Emergencia_OP10_OK )
      Coil( %DB12.DBX1.1 )
   END_RUNG
   // the same network as SCL:
   %DB12.DBX1.1 := NOT "Multiplo_Uso_DB".Emergencia_OP10_OK;
END_REGION

REGION Network 3
   RUNG wire#powerrail
      I_Contact( "Multiplo_Uso_DB".Emergencia_OP20_OK )
      Coil( %DB12.DBX1.2 )
   END_RUNG
   // the same network as SCL:
   %DB12.DBX1.2 := NOT "Multiplo_Uso_DB".Emergencia_OP20_OK;
END_REGION

REGION Network 4
   RUNG wire#powerrail
      I_Contact( "Multiplo_Uso_DB".Emergencia_OP30_OK )
      Coil( %DB12.DBX1.3 )
   END_RUNG
   // the same network as SCL:
   %DB12.DBX1.3 := NOT "Multiplo_Uso_DB".Emergencia_OP30_OK;
END_REGION

REGION Network 5
   RUNG wire#powerrail
      I_Contact( "Multiplo_Uso_DB".Emergencia_OP40_OK )
      Coil( %DB12.DBX1.4 )
   END_RUNG
   // the same network as SCL:
   %DB12.DBX1.4 := NOT "Multiplo_Uso_DB".Emergencia_OP40_OK;
END_REGION

REGION Network 6
   RUNG wire#powerrail
      Contact( "Multiplo_Uso_DB".Emergencia_OP50_OK )
      Coil( %DB12.DBX1.5 )
   END_RUNG
   // the same network as SCL:
   %DB12.DBX1.5 := "Multiplo_Uso_DB".Emergencia_OP50_OK;
END_REGION

REGION Network 7
   RUNG wire#powerrail
      Contact( "Multiplo_Uso_DB".Emergencia_OP60_OK )
      Coil( %DB12.DBX1.6 )
   END_RUNG
   // the same network as SCL:
   %DB12.DBX1.6 := "Multiplo_Uso_DB".Emergencia_OP60_OK;
END_REGION

REGION Network 8
   RUNG wire#powerrail
      Contact( "Multiplo_Uso_DB".Emergencia_OP70_OK )
      Coil( %DB12.DBX1.7 )
   END_RUNG
   // the same network as SCL:
   %DB12.DBX1.7 := "Multiplo_Uso_DB".Emergencia_OP70_OK;
END_REGION

REGION Network 9
   RUNG wire#powerrail
      Contact( "Multiplo_Uso_DB".Emergencia_OP80_OK )
      Coil( %DB12.DBX0.0 )
   END_RUNG
   // the same network as SCL:
   %DB12.DBX0.0 := "Multiplo_Uso_DB".Emergencia_OP80_OK;
END_REGION

REGION Network 10
   RUNG wire#powerrail
      I_Contact( "12ME02_Termostato¶Painel" )
      Coil( %DB12.DBX0.1 )
   END_RUNG
   // the same network as SCL:
   %DB12.DBX0.1 := NOT "12ME02_Termostato¶Painel";
END_REGION

REGION Network 11
   RUNG wire#powerrail
      I_Contact( "12ME02_Disjuntor¶Serviço Ok" )
      Coil( %DB12.DBX0.2 )
   END_RUNG
   // the same network as SCL:
   %DB12.DBX0.2 := NOT "12ME02_Disjuntor¶Serviço Ok";
END_REGION

REGION Network 12
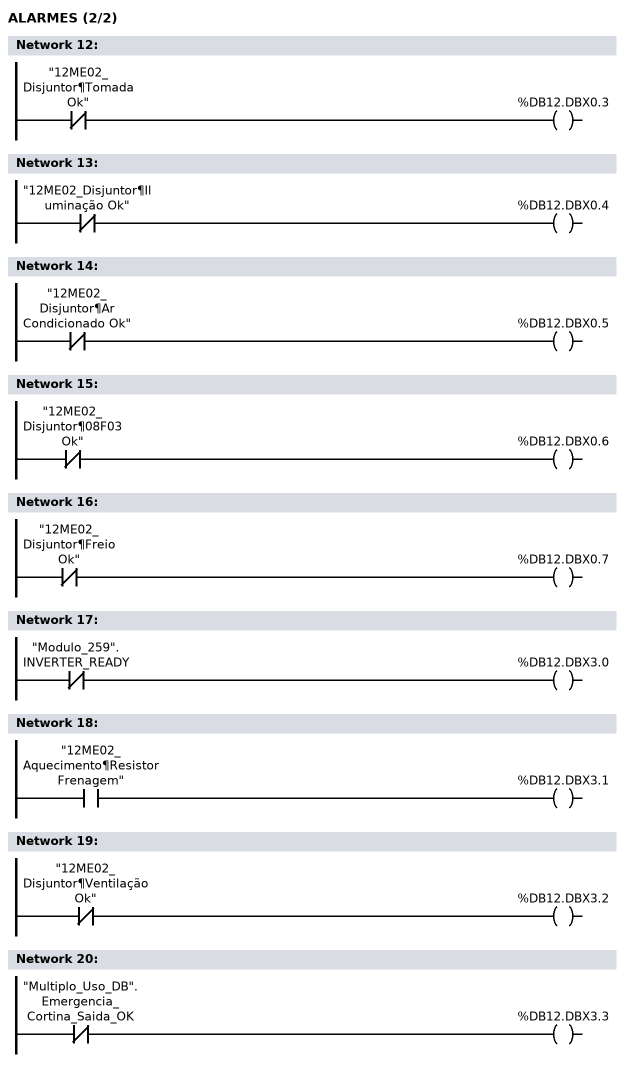
   RUNG wire#powerrail
      I_Contact( "12ME02_Disjuntor¶Tomada Ok" )
      Coil( %DB12.DBX0.3 )
   END_RUNG
   // the same network as SCL:
   %DB12.DBX0.3 := NOT "12ME02_Disjuntor¶Tomada Ok";
END_REGION

REGION Network 13
   RUNG wire#powerrail
      I_Contact( "12ME02_Disjuntor¶Iluminação Ok" )
      Coil( %DB12.DBX0.4 )
   END_RUNG
   // the same network as SCL:
   %DB12.DBX0.4 := NOT "12ME02_Disjuntor¶Iluminação Ok";
END_REGION

REGION Network 14
   RUNG wire#powerrail
      I_Contact( "12ME02_Disjuntor¶Ar Condicionado Ok" )
      Coil( %DB12.DBX0.5 )
   END_RUNG
   // the same network as SCL:
   %DB12.DBX0.5 := NOT "12ME02_Disjuntor¶Ar Condicionado Ok";
END_REGION

REGION Network 15
   RUNG wire#powerrail
      I_Contact( "12ME02_Disjuntor¶08F03 Ok" )
      Coil( %DB12.DBX0.6 )
   END_RUNG
   // the same network as SCL:
   %DB12.DBX0.6 := NOT "12ME02_Disjuntor¶08F03 Ok";
END_REGION

REGION Network 16
   RUNG wire#powerrail
      I_Contact( "12ME02_Disjuntor¶Freio Ok" )
      Coil( %DB12.DBX0.7 )
   END_RUNG
   // the same network as SCL:
   %DB12.DBX0.7 := NOT "12ME02_Disjuntor¶Freio Ok";
END_REGION

REGION Network 17
   RUNG wire#powerrail
      I_Contact( "Modulo_259".INVERTER_READY )
      Coil( %DB12.DBX3.0 )
   END_RUNG
   // the same network as SCL:
   %DB12.DBX3.0 := NOT "Modulo_259".INVERTER_READY;
END_REGION

REGION Network 18
   RUNG wire#powerrail
      Contact( "12ME02_Aquecimento¶Resistor Frenagem" )
      Coil( %DB12.DBX3.1 )
   END_RUNG
   // the same network as SCL:
   %DB12.DBX3.1 := "12ME02_Aquecimento¶Resistor Frenagem";
END_REGION

REGION Network 19
   RUNG wire#powerrail
      I_Contact( "12ME02_Disjuntor¶Ventilação Ok" )
      Coil( %DB12.DBX3.2 )
   END_RUNG
   // the same network as SCL:
   %DB12.DBX3.2 := NOT "12ME02_Disjuntor¶Ventilação Ok";
END_REGION

REGION Network 20
   RUNG wire#powerrail
      I_Contact( "Multiplo_Uso_DB".Emergencia_Cortina_Saida_OK )
      Coil( %DB12.DBX3.3 )
   END_RUNG
   // the same network as SCL:
   %DB12.DBX3.3 := NOT "Multiplo_Uso_DB".Emergencia_Cortina_Saida_OK;
END_REGION
END_FUNCTION

FUNCTION "CONTROLES_SISTEMA" : Void   // FC3, LAD
{ S7_Optimized_Access := 'TRUE' }
VERSION : 0.1
   VAR_TEMP   // added for the SCL form of the ladder/FBD networks
      _w1 : Bool;
   END_VAR
BEGIN

REGION Network 1: lIGA AUTOMATICO/MANUAL
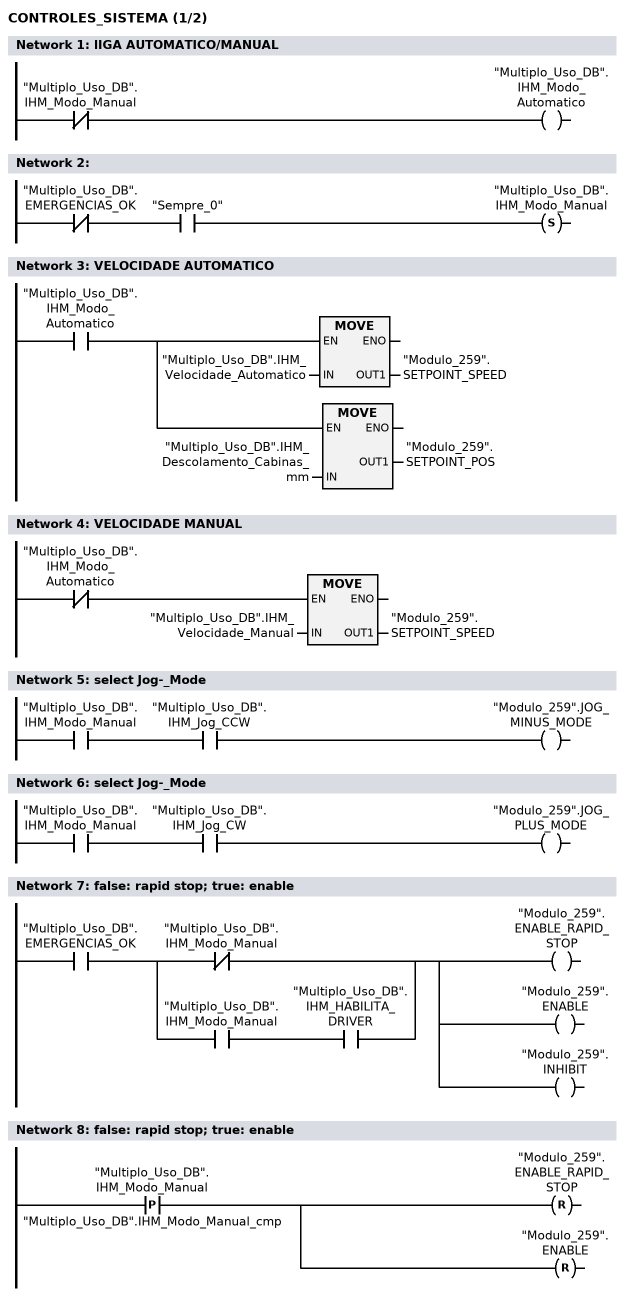
   RUNG wire#powerrail
      I_Contact( "Multiplo_Uso_DB".IHM_Modo_Manual )
      Coil( "Multiplo_Uso_DB".IHM_Modo_Automatico )
   END_RUNG
   // the same network as SCL:
   "Multiplo_Uso_DB".IHM_Modo_Automatico := NOT "Multiplo_Uso_DB".IHM_Modo_Manual;
END_REGION

REGION Network 2
   RUNG wire#powerrail
      I_Contact( "Multiplo_Uso_DB".EMERGENCIAS_OK )
      Contact( "Sempre_0" )
      S_Coil( "Multiplo_Uso_DB".IHM_Modo_Manual )
   END_RUNG
   // the same network as SCL:
   IF NOT "Multiplo_Uso_DB".EMERGENCIAS_OK AND "Sempre_0" THEN
       "Multiplo_Uso_DB".IHM_Modo_Manual := TRUE;
   END_IF;
END_REGION

REGION Network 3: VELOCIDADE AUTOMATICO
   RUNG wire#powerrail
      Contact( "Multiplo_Uso_DB".IHM_Modo_Automatico )
      wire#w1
      Move(in := "Multiplo_Uso_DB".IHM_Velocidade_Automatico, out1 => "Modulo_259".SETPOINT_SPEED)
   END_RUNG
   RUNG wire#w1
      Move(in := "Multiplo_Uso_DB".IHM_Descolamento_Cabinas_mm, out1 => "Modulo_259".SETPOINT_POS)
   END_RUNG
   // the same network as SCL:
   IF "Multiplo_Uso_DB".IHM_Modo_Automatico THEN
       "Modulo_259".SETPOINT_SPEED := "Multiplo_Uso_DB".IHM_Velocidade_Automatico;
       "Modulo_259".SETPOINT_POS := "Multiplo_Uso_DB".IHM_Descolamento_Cabinas_mm;
   END_IF;
END_REGION

REGION Network 4: VELOCIDADE MANUAL
   RUNG wire#powerrail
      I_Contact( "Multiplo_Uso_DB".IHM_Modo_Automatico )
      Move(in := "Multiplo_Uso_DB".IHM_Velocidade_Manual, out1 => "Modulo_259".SETPOINT_SPEED)
   END_RUNG
   // the same network as SCL:
   IF NOT "Multiplo_Uso_DB".IHM_Modo_Automatico THEN
       "Modulo_259".SETPOINT_SPEED := "Multiplo_Uso_DB".IHM_Velocidade_Manual;
   END_IF;
END_REGION

REGION Network 5: select Jog-_Mode
   RUNG wire#powerrail
      Contact( "Multiplo_Uso_DB".IHM_Modo_Manual )
      Contact( "Multiplo_Uso_DB".IHM_Jog_CCW )
      Coil( "Modulo_259".JOG_MINUS_MODE )
   END_RUNG
   // the same network as SCL:
   "Modulo_259".JOG_MINUS_MODE := "Multiplo_Uso_DB".IHM_Modo_Manual AND "Multiplo_Uso_DB".IHM_Jog_CCW;
END_REGION

REGION Network 6: select Jog-_Mode
   RUNG wire#powerrail
      Contact( "Multiplo_Uso_DB".IHM_Modo_Manual )
      Contact( "Multiplo_Uso_DB".IHM_Jog_CW )
      Coil( "Modulo_259".JOG_PLUS_MODE )
   END_RUNG
   // the same network as SCL:
   "Modulo_259".JOG_PLUS_MODE := "Multiplo_Uso_DB".IHM_Modo_Manual AND "Multiplo_Uso_DB".IHM_Jog_CW;
END_REGION

REGION Network 7: false: rapid stop; true: enable
   RUNG wire#powerrail
      Contact( "Multiplo_Uso_DB".EMERGENCIAS_OK )
      wire#w1
      I_Contact( "Multiplo_Uso_DB".IHM_Modo_Manual )
      wire#w2
      Coil( "Modulo_259".ENABLE_RAPID_STOP )
   END_RUNG
   RUNG wire#w1
      Contact( "Multiplo_Uso_DB".IHM_Modo_Manual )
      Contact( "Multiplo_Uso_DB".IHM_HABILITA_DRIVER )
   END_RUNG wire#w2
   RUNG wire#w2
      Coil( "Modulo_259".ENABLE )
   END_RUNG
   RUNG wire#w2
      Coil( "Modulo_259".INHIBIT )
   END_RUNG
   // the same network as SCL:
   "Modulo_259".ENABLE_RAPID_STOP := "Multiplo_Uso_DB".EMERGENCIAS_OK AND (NOT "Multiplo_Uso_DB".IHM_Modo_Manual OR ("Multiplo_Uso_DB".IHM_Modo_Manual AND "Multiplo_Uso_DB".IHM_HABILITA_DRIVER));
   "Modulo_259".ENABLE := "Modulo_259".ENABLE_RAPID_STOP;
   "Modulo_259".INHIBIT := "Modulo_259".ENABLE_RAPID_STOP;
END_REGION

REGION Network 8: false: rapid stop; true: enable
   RUNG wire#powerrail
      P_Contact(operand := "Multiplo_Uso_DB".IHM_Modo_Manual, bit := "Multiplo_Uso_DB".IHM_Modo_Manual_cmp)
      wire#w1
      R_Coil( "Modulo_259".ENABLE_RAPID_STOP )
   END_RUNG
   RUNG wire#w1
      R_Coil( "Modulo_259".ENABLE )
   END_RUNG
   // the same network as SCL:
   #_w1 := "Multiplo_Uso_DB".IHM_Modo_Manual AND NOT "Multiplo_Uso_DB".IHM_Modo_Manual_cmp;   // rising edge of "Multiplo_Uso_DB".IHM_Modo_Manual
   "Multiplo_Uso_DB".IHM_Modo_Manual_cmp := "Multiplo_Uso_DB".IHM_Modo_Manual;
   IF #_w1 THEN
       "Modulo_259".ENABLE_RAPID_STOP := FALSE;
       "Modulo_259".ENABLE := FALSE;
   END_IF;
END_REGION

REGION Network 9: DRIVER MODO AUTOMATICO
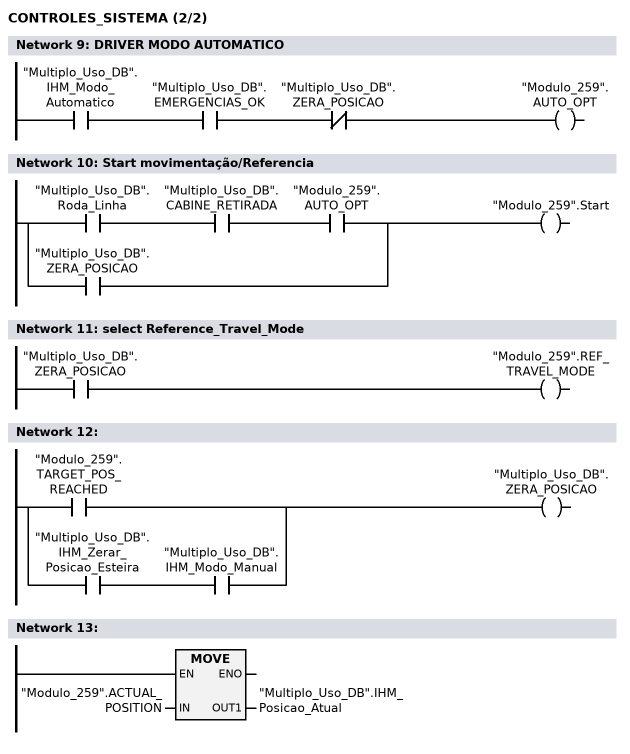
   RUNG wire#powerrail
      Contact( "Multiplo_Uso_DB".IHM_Modo_Automatico )
      Contact( "Multiplo_Uso_DB".EMERGENCIAS_OK )
      I_Contact( "Multiplo_Uso_DB".ZERA_POSICAO )
      Coil( "Modulo_259".AUTO_OPT )
   END_RUNG
   // the same network as SCL:
   "Modulo_259".AUTO_OPT := "Multiplo_Uso_DB".IHM_Modo_Automatico AND "Multiplo_Uso_DB".EMERGENCIAS_OK AND NOT "Multiplo_Uso_DB".ZERA_POSICAO;
END_REGION

REGION Network 10: Start movimentação/Referencia
   RUNG wire#powerrail
      Contact( "Multiplo_Uso_DB".Roda_Linha )
      Contact( "Multiplo_Uso_DB".CABINE_RETIRADA )
      Contact( "Modulo_259".AUTO_OPT )
      wire#w1
      Coil( "Modulo_259".Start )
   END_RUNG
   RUNG wire#powerrail
      Contact( "Multiplo_Uso_DB".ZERA_POSICAO )
   END_RUNG wire#w1
   // the same network as SCL:
   "Modulo_259".Start := ("Multiplo_Uso_DB".Roda_Linha AND "Multiplo_Uso_DB".CABINE_RETIRADA AND "Modulo_259".AUTO_OPT) OR "Multiplo_Uso_DB".ZERA_POSICAO;
END_REGION

REGION Network 11: select Reference_Travel_Mode
   RUNG wire#powerrail
      Contact( "Multiplo_Uso_DB".ZERA_POSICAO )
      Coil( "Modulo_259".REF_TRAVEL_MODE )
   END_RUNG
   // the same network as SCL:
   "Modulo_259".REF_TRAVEL_MODE := "Multiplo_Uso_DB".ZERA_POSICAO;
END_REGION

REGION Network 12
   RUNG wire#powerrail
      Contact( "Modulo_259".TARGET_POS_REACHED )
      wire#w1
      Coil( "Multiplo_Uso_DB".ZERA_POSICAO )
   END_RUNG
   RUNG wire#powerrail
      Contact( "Multiplo_Uso_DB".IHM_Zerar_Posicao_Esteira )
      Contact( "Multiplo_Uso_DB".IHM_Modo_Manual )
   END_RUNG wire#w1
   // the same network as SCL:
   "Multiplo_Uso_DB".ZERA_POSICAO := "Modulo_259".TARGET_POS_REACHED OR ("Multiplo_Uso_DB".IHM_Zerar_Posicao_Esteira AND "Multiplo_Uso_DB".IHM_Modo_Manual);
END_REGION

REGION Network 13
   RUNG wire#powerrail
      Move(in := "Modulo_259".ACTUAL_POSITION, out1 => "Multiplo_Uso_DB".IHM_Posicao_Atual)
   END_RUNG
   // the same network as SCL:
   "Multiplo_Uso_DB".IHM_Posicao_Atual := "Modulo_259".ACTUAL_POSITION;
END_REGION
END_FUNCTION

FUNCTION "Dados_Andon" : Void   // FC4, LAD
{ S7_Optimized_Access := 'TRUE' }
VERSION : 0.1
   VAR_TEMP
      move_dados : Bool;
      move_dados_cmp : Bool;
   END_VAR
BEGIN

REGION Network 1: Contagem cabinas
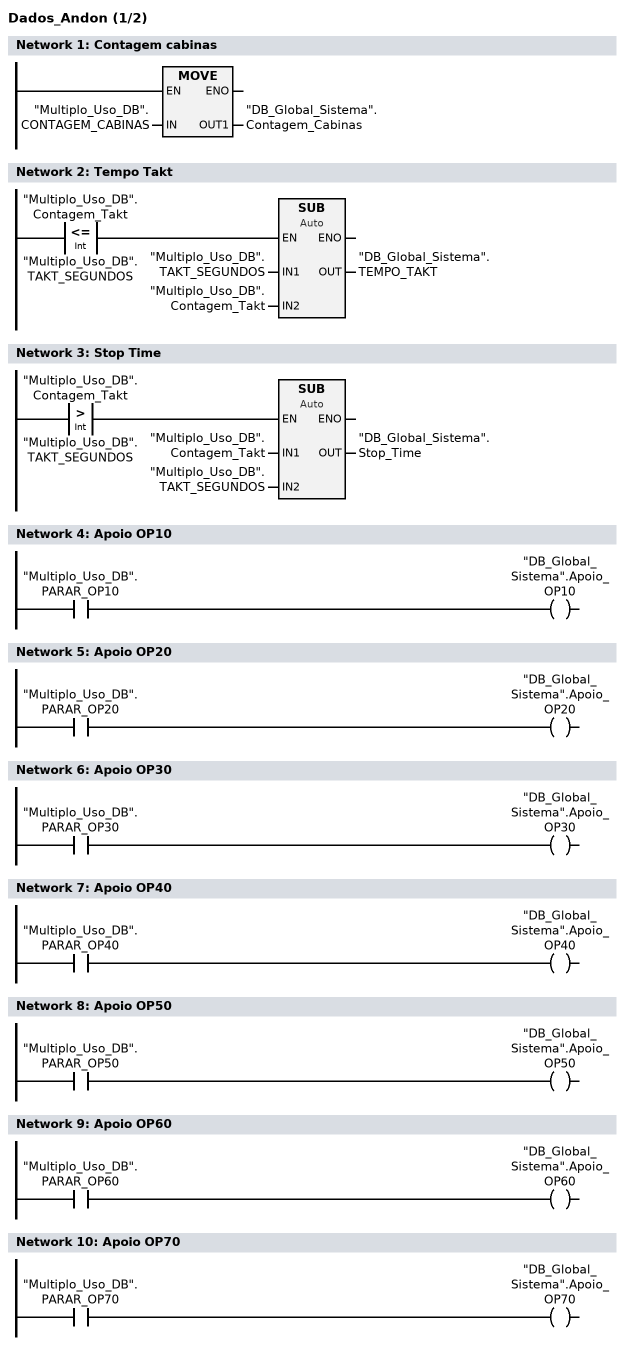
   RUNG wire#powerrail
      Move(in := "Multiplo_Uso_DB".CONTAGEM_CABINAS, out1 => "DB_Global_Sistema".Contagem_Cabinas)
   END_RUNG
   // the same network as SCL:
   "DB_Global_Sistema".Contagem_Cabinas := "Multiplo_Uso_DB".CONTAGEM_CABINAS;
END_REGION

REGION Network 2: Tempo Takt
   RUNG wire#powerrail
      { S7_Templates := "SrcType := Int" } LE_Contact(in1 := "Multiplo_Uso_DB".Contagem_Takt, in2 := "Multiplo_Uso_DB".TAKT_SEGUNDOS)
      Sub(in1 := "Multiplo_Uso_DB".TAKT_SEGUNDOS, in2 := "Multiplo_Uso_DB".Contagem_Takt, out => "DB_Global_Sistema".TEMPO_TAKT)
   END_RUNG
   // the same network as SCL:
   IF "Multiplo_Uso_DB".Contagem_Takt <= "Multiplo_Uso_DB".TAKT_SEGUNDOS THEN
       "DB_Global_Sistema".TEMPO_TAKT := "Multiplo_Uso_DB".TAKT_SEGUNDOS - "Multiplo_Uso_DB".Contagem_Takt;
   END_IF;
END_REGION

REGION Network 3: Stop Time
   RUNG wire#powerrail
      { S7_Templates := "SrcType := Int" } GT_Contact(in1 := "Multiplo_Uso_DB".Contagem_Takt, in2 := "Multiplo_Uso_DB".TAKT_SEGUNDOS)
      Sub(in1 := "Multiplo_Uso_DB".Contagem_Takt, in2 := "Multiplo_Uso_DB".TAKT_SEGUNDOS, out => "DB_Global_Sistema".Stop_Time)
   END_RUNG
   // the same network as SCL:
   IF "Multiplo_Uso_DB".Contagem_Takt > "Multiplo_Uso_DB".TAKT_SEGUNDOS THEN
       "DB_Global_Sistema".Stop_Time := "Multiplo_Uso_DB".Contagem_Takt - "Multiplo_Uso_DB".TAKT_SEGUNDOS;
   END_IF;
END_REGION

REGION Network 4: Apoio OP10
   RUNG wire#powerrail
      Contact( "Multiplo_Uso_DB".PARAR_OP10 )
      Coil( "DB_Global_Sistema".Apoio_OP10 )
   END_RUNG
   // the same network as SCL:
   "DB_Global_Sistema".Apoio_OP10 := "Multiplo_Uso_DB".PARAR_OP10;
END_REGION

REGION Network 5: Apoio OP20
   RUNG wire#powerrail
      Contact( "Multiplo_Uso_DB".PARAR_OP20 )
      Coil( "DB_Global_Sistema".Apoio_OP20 )
   END_RUNG
   // the same network as SCL:
   "DB_Global_Sistema".Apoio_OP20 := "Multiplo_Uso_DB".PARAR_OP20;
END_REGION

REGION Network 6: Apoio OP30
   RUNG wire#powerrail
      Contact( "Multiplo_Uso_DB".PARAR_OP30 )
      Coil( "DB_Global_Sistema".Apoio_OP30 )
   END_RUNG
   // the same network as SCL:
   "DB_Global_Sistema".Apoio_OP30 := "Multiplo_Uso_DB".PARAR_OP30;
END_REGION

REGION Network 7: Apoio OP40
   RUNG wire#powerrail
      Contact( "Multiplo_Uso_DB".PARAR_OP40 )
      Coil( "DB_Global_Sistema".Apoio_OP40 )
   END_RUNG
   // the same network as SCL:
   "DB_Global_Sistema".Apoio_OP40 := "Multiplo_Uso_DB".PARAR_OP40;
END_REGION

REGION Network 8: Apoio OP50
   RUNG wire#powerrail
      Contact( "Multiplo_Uso_DB".PARAR_OP50 )
      Coil( "DB_Global_Sistema".Apoio_OP50 )
   END_RUNG
   // the same network as SCL:
   "DB_Global_Sistema".Apoio_OP50 := "Multiplo_Uso_DB".PARAR_OP50;
END_REGION

REGION Network 9: Apoio OP60
   RUNG wire#powerrail
      Contact( "Multiplo_Uso_DB".PARAR_OP60 )
      Coil( "DB_Global_Sistema".Apoio_OP60 )
   END_RUNG
   // the same network as SCL:
   "DB_Global_Sistema".Apoio_OP60 := "Multiplo_Uso_DB".PARAR_OP60;
END_REGION

REGION Network 10: Apoio OP70
   RUNG wire#powerrail
      Contact( "Multiplo_Uso_DB".PARAR_OP70 )
      Coil( "DB_Global_Sistema".Apoio_OP70 )
   END_RUNG
   // the same network as SCL:
   "DB_Global_Sistema".Apoio_OP70 := "Multiplo_Uso_DB".PARAR_OP70;
END_REGION

REGION Network 11: Apoio OP80
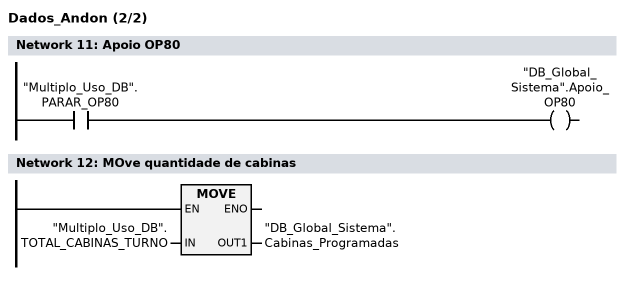
   RUNG wire#powerrail
      Contact( "Multiplo_Uso_DB".PARAR_OP80 )
      Coil( "DB_Global_Sistema".Apoio_OP80 )
   END_RUNG
   // the same network as SCL:
   "DB_Global_Sistema".Apoio_OP80 := "Multiplo_Uso_DB".PARAR_OP80;
END_REGION

REGION Network 12: MOve quantidade de cabinas
   RUNG wire#powerrail
      Move(in := "Multiplo_Uso_DB".TOTAL_CABINAS_TURNO, out1 => "DB_Global_Sistema".Cabinas_Programadas)
   END_RUNG
   // the same network as SCL:
   "DB_Global_Sistema".Cabinas_Programadas := "Multiplo_Uso_DB".TOTAL_CABINAS_TURNO;
END_REGION
END_FUNCTION

FUNCTION "call_Modulo" : Void   // FC100, FBD
TITLE = Call Modulo Positioning
{ S7_Optimized_Access := 'TRUE' }
VERSION : 0.2
// Comment:
// This sample program shows the basic approach only.
// We do not accept legal or other liability for
// incorrect program functions and their consequences!
BEGIN

REGION Network 1: Call Modulo Positioning (PROFINET IO)
   // Startup the MOVIDRIVE Application Module "Modulo Posi."
   // 
   // Attention: "IO_ADDRESS_or_HW_IDENTIFIER"
   // S73xx/4xx: Assign Peripheral Address; S7 1x00: assign HW_Identifier
   // 
   // The FC141 serve as sample program element for control of the 
   // application module "MODULO pOSI" for units of the 
   // MOVIDRIVE series in technology variants.
   // 
   // The FC141 can be used to control the drive inverter via PROFIBUS DP or PROFINET 
   // IO. 
   // 
   // You display the process data in the bus positioning monitor 
   // after startup of the application module. You will find additional 
   // information, such as coding of the process data, in the MOTIONSTUDIO online help.
   // 
   // FC inputs:
   // "INHIBIT" = true: enable; false: inhibit
   // "ENABLE_RAPID_STOP" = true: Enable; false: Rapid stop
   // "ENABLE" = true: enable; false: STOP
   // "RESET": Confirm error
   // "Start": Movement takes place to the specified target position when "Start" is set and the unit status is the technology function
   // Select the operating mode with the inputs "Jog_plus_mode, Jog_minus_mode; 
   // Ref_travel, Auto,..,..
   // "SETPOINT_POS": Position setpoint (DINT) in user unit.
   // The user unit depends on the startup of the "Modulo Posi.."
   // "SETPOINT_SPEED": Positioning speed (INT) in rpm
   // "START_RAMP": Acceleration ramp (INT) in ms
   // "STOP_RAMP": Deceleration ramp(INT) in ms
   // 
   // FC outputs:
   // If the data transmission/PROFIBUS is disrupted, all outputs will be deleted.
   // => "COMMUNICATION_OK = false (self-confirming)
   // "FAULT_OF_AXIS" = true: An error is present.
   // "WARNING_OF_AXIS" = true: A warning is present.
   // "INVERTER_READY" = true: There is no error & mains voltage ON"
   // "REFERENCED" = true: The axis is referenced 
   // TARGET_POS_REACHED" = true: Target position has been reached.
   // "AXIS_INTERLOCKED" = true: Reports back that there is an illogical mode 
   // selection. (=> none or several modes selected)
   // "FAULT_NO" <> 0: The error codes are listed in the system manual and are 
   // displayed in MOVITOOLS (status, bus monitor).
   // "ACTUAL_POSITION": Actual position (DINT) in user unit.
   // "ACTUAL_SPEED": Actual speed (INT) in rpm
   // "ACTUAL_CURRENT": Actual current (effective current) as percentage of rated 
   // unit current
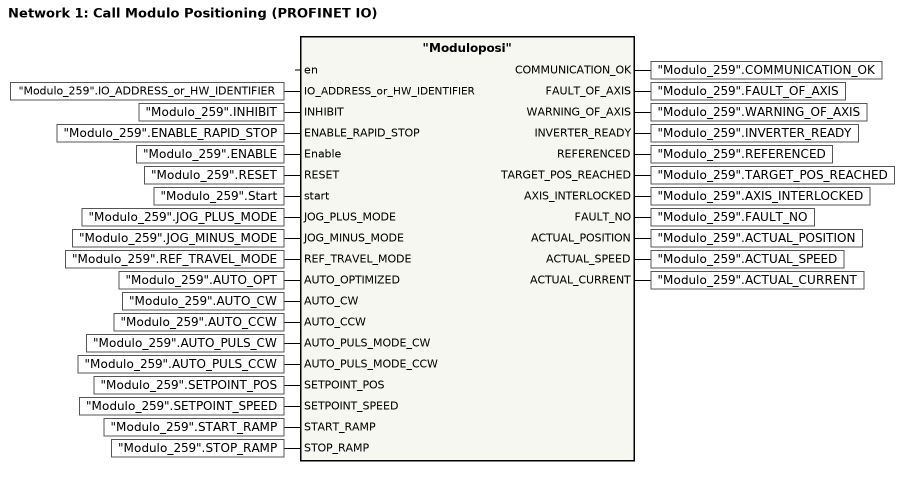
   "Moduloposi"(IO_ADDRESS_or_HW_IDENTIFIER := "Modulo_259".IO_ADDRESS_or_HW_IDENTIFIER,
                INHIBIT := "Modulo_259".INHIBIT,
                ENABLE_RAPID_STOP := "Modulo_259".ENABLE_RAPID_STOP,
                Enable := "Modulo_259".ENABLE,
                RESET := "Modulo_259".RESET,
                start := "Modulo_259".Start,
                JOG_PLUS_MODE := "Modulo_259".JOG_PLUS_MODE,
                JOG_MINUS_MODE := "Modulo_259".JOG_MINUS_MODE,
                REF_TRAVEL_MODE := "Modulo_259".REF_TRAVEL_MODE,
                AUTO_OPTIMIZED := "Modulo_259".AUTO_OPT,
                AUTO_CW := "Modulo_259".AUTO_CW,
                AUTO_CCW := "Modulo_259".AUTO_CCW,
                AUTO_PULS_MODE_CW := "Modulo_259".AUTO_PULS_CW,
                AUTO_PULS_MODE_CCW := "Modulo_259".AUTO_PULS_CCW,
                SETPOINT_POS := "Modulo_259".SETPOINT_POS,
                SETPOINT_SPEED := "Modulo_259".SETPOINT_SPEED,
                START_RAMP := "Modulo_259".START_RAMP,
                STOP_RAMP := "Modulo_259".STOP_RAMP,
                COMMUNICATION_OK => "Modulo_259".COMMUNICATION_OK,
                FAULT_OF_AXIS => "Modulo_259".FAULT_OF_AXIS,
                WARNING_OF_AXIS => "Modulo_259".WARNING_OF_AXIS,
                INVERTER_READY => "Modulo_259".INVERTER_READY,
                REFERENCED => "Modulo_259".REFERENCED,
                TARGET_POS_REACHED => "Modulo_259".TARGET_POS_REACHED,
                AXIS_INTERLOCKED => "Modulo_259".AXIS_INTERLOCKED,
                FAULT_NO => "Modulo_259".FAULT_NO,
                ACTUAL_POSITION => "Modulo_259".ACTUAL_POSITION,
                ACTUAL_SPEED => "Modulo_259".ACTUAL_SPEED,
                ACTUAL_CURRENT => "Modulo_259".ACTUAL_CURRENT);
END_REGION
END_FUNCTION

FUNCTION "Moduloposi" : Void   // FC141, FBD
TITLE = Modulopos
{ S7_Optimized_Access := 'FALSE' }
AUTHOR : BUCPAEM
FAMILY : PROFIBUS
NAME : MDX_POS
VERSION : 0.1
// This sample program shows the basic approach only.
// We do not accept legal or other liability for
// incorrect program functions and their consequences!
// Dieses Programmbeispiel zeigt nur die prinzipielle Vorgehensweise.
// Für fehlerhafte Programmfunktionen und deren Folgen
// kann weder eine juristische, noch irgendeine Haftung übernommen werden!
   VAR_INPUT
      IO_ADDRESS_or_HW_IDENTIFIER : Hw_Io;   // S71xxxx: assign HW_Identifier; S74xx/3xx assign Peripheral address
      INHIBIT : Bool;   // false: Contr. inhibit; true: enable
      ENABLE_RAPID_STOP : Bool;   // false: rapid stop; true: enable
      Enable : Bool;   // false: stop; true: enable
      RESET : Bool;
      start : Bool;
      JOG_PLUS_MODE : Bool;   // select Jog+_Mode
      JOG_MINUS_MODE : Bool;   // select Jog-_Mode
      REF_TRAVEL_MODE : Bool;   // REF_TRAVEL_MODE angewählt
      AUTO_OPTIMIZED : Bool;   // select AUTO_OPT_Mode
      AUTO_CW : Bool;   // select AUTO_CW_Mode
      AUTO_CCW : Bool;   // select AUTO_CCW_Mode
      AUTO_PULS_MODE_CW : Bool;   // select AUTO_PULS_CW_Mode
      AUTO_PULS_MODE_CCW : Bool;   // select AUTO_PULS_CCW_Mode
      SETPOINT_POS : DInt;
      SETPOINT_SPEED : Int;
      START_RAMP : Int;   // Attention: Avoid Ramp = 0!
      STOP_RAMP : Int;   // Attention: Avoid Ramp = 0!
   END_VAR
   VAR_OUTPUT
      COMMUNICATION_OK : Bool;   // DPRD_DAT & DPWR_DAT: Return Value = 0 / SFC14/SFC15: Return Value = 0
      FAULT_OF_AXIS : Bool;   // A fault is active, if the inverter is not ready for operation AND the error bit has been set.
      WARNING_OF_AXIS : Bool;   // A warning is active, if the inverter is still ready for operation AND the error bit has been set.
      INVERTER_READY : Bool;
      REFERENCED : Bool;
      TARGET_POS_REACHED : Bool;
      AXIS_INTERLOCKED : Bool;   // mode selection is illogical (no mode or several modes selected) / die Modeanwahl ist unplausibel (kein Mode oder mehrere Modi angewählt)
      FAULT_NO : Int;
      ACTUAL_POSITION : DInt;
      ACTUAL_SPEED : Int;
      ACTUAL_CURRENT : Int;
   END_VAR
   VAR_TEMP
      PI : Struct   // Prozeßeingangsdaten
         Status : Byte;
         Motor_turning : Bool;
         Inverter_ready : Bool;
         referenced : Bool;
         Target_position_reached : Bool;
         Brake_released : Bool;
         Error : Bool;
         reserved_Bit_14 : Bool;
         reserved_Bit_15 : Bool;
         Actual_position : DInt;
         Actual_speed : Int;
         Active_current : Int;
         Device_utilisation : Int;
      END_STRUCT;
      PO : Struct   // Prozeßausgangsdaten
         start : Bool;
         Jog_plus : Bool;
         Jog_minus : Bool;
         mode_Bit11 : Bool;
         mode_Bit12 : Bool;
         mode_Bit13 : Bool;
         CTW_Bit_14 : Bool;
         CTW_Bit_15 : Bool;
         Contr_inhibit : Bool;
         Rapid_stop : Bool;
         Stop : Bool;
         CTW_Bit_3 : Bool;
         CTW_Bit_4 : Bool;
         CTW_Bit_5 : Bool;
         Reset_fault : Bool;
         CTW_Bit_7 : Bool;
         Setpoint_position : DInt;
         Setpoint_speed : Int;
         Start_ramp : Int;
         Stop_ramp : Int;
      END_STRUCT;
      tRef : Bool;
      tAuto_opti : Bool;
      tAuto_CW : Bool;
      tAuto_CCW : Bool;
      tAUTO_PULS_MODE_CW : Bool;
      tAUTO_PULS_MODE_CCW : Bool;
      FALSE : Bool;
      Addr : Word;
      Returncode_SFC14 : Int;
      Returncode_SFC15 : Int;
      Com_SFC14_OK : Bool;
      Com_SFC15_OK : Bool;
   END_VAR
   VAR_TEMP   // added for the SCL form of the ladder/FBD networks
      _w1 : Bool;
   END_VAR
BEGIN

REGION Network 1: Def. "#FALSE"
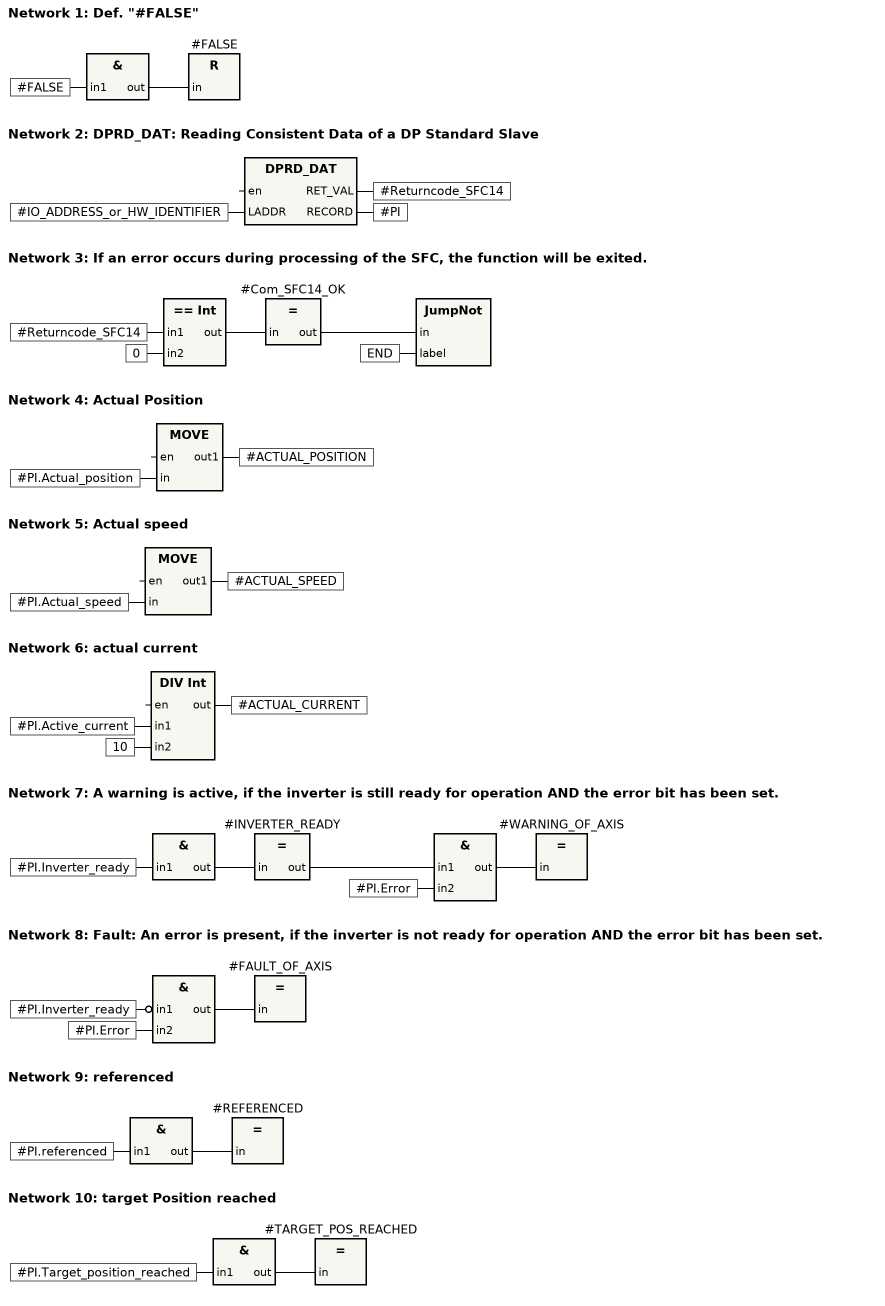
   IF #FALSE THEN #FALSE := FALSE; END_IF;
END_REGION

REGION Network 2: DPRD_DAT: Reading Consistent Data of a DP Standard Slave
   #Returncode_SFC14 := DPRD_DAT(LADDR := #IO_ADDRESS_or_HW_IDENTIFIER, RECORD => #PI);
END_REGION

REGION Network 3: If an error occurs during processing of the SFC, the function will be exited.
   // no SCL statement known for JumpNot: written as a call
   #Com_SFC14_OK := #Returncode_SFC14 = 0;
   JumpNot(in := #Com_SFC14_OK, label := END);
END_REGION

REGION Network 4: Actual Position
   #ACTUAL_POSITION := #PI.Actual_position;
END_REGION

REGION Network 5: Actual speed
   #ACTUAL_SPEED := #PI.Actual_speed;
END_REGION

REGION Network 6: actual current
   #ACTUAL_CURRENT := #PI.Active_current / 10;
END_REGION

REGION Network 7: A warning is active, if the inverter is still ready for operation AND the error bit has been set.
   #INVERTER_READY := #PI.Inverter_ready;
   #WARNING_OF_AXIS := #PI.Inverter_ready AND #PI.Error;
END_REGION

REGION Network 8: Fault: An error is present, if the inverter is not ready for operation AND the error bit has been set.
   #FAULT_OF_AXIS := NOT #PI.Inverter_ready AND #PI.Error;
END_REGION

REGION Network 9: referenced
   #REFERENCED := #PI.referenced;
END_REGION

REGION Network 10: target Position reached
   #TARGET_POS_REACHED := #PI.Target_position_reached;
END_REGION

REGION Network 11: Fault_NO
   // If Error is true => Fault_NO := High Byte of the Status word
   // If Error is false => Fault_NO := 0
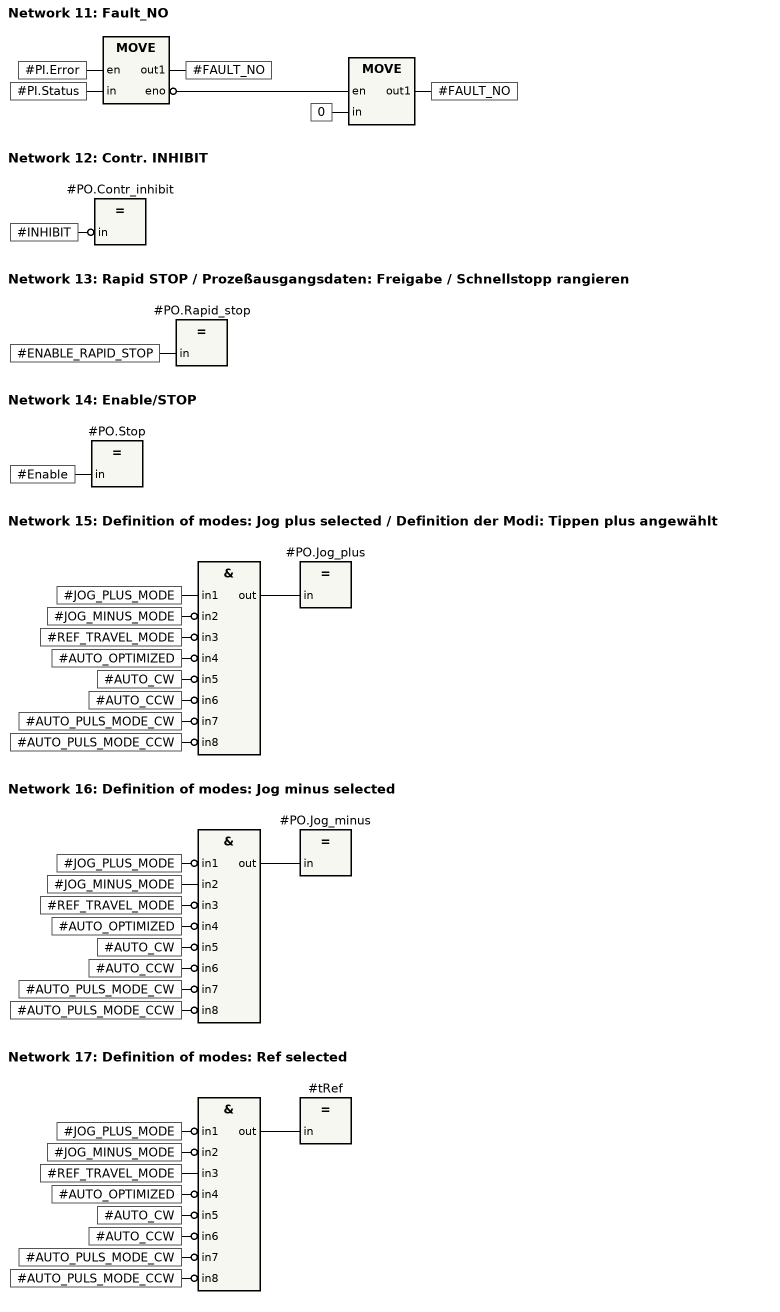
   // ENO of a box is taken as its EN; it also drops when the box reports an error
   IF #PI.Error THEN #FAULT_NO := #PI.Status; END_IF;
   IF NOT #PI.Error THEN #FAULT_NO := 0; END_IF;
END_REGION

REGION Network 12: Contr. INHIBIT
   #PO.Contr_inhibit := NOT #INHIBIT;
END_REGION

REGION Network 13: Rapid STOP / Prozeßausgangsdaten: Freigabe / Schnellstopp rangieren
   #PO.Rapid_stop := #ENABLE_RAPID_STOP;
END_REGION

REGION Network 14: Enable/STOP
   #PO.Stop := #Enable;
END_REGION

REGION Network 15: Definition of modes: Jog plus selected / Definition der Modi: Tippen plus angewählt
   #PO.Jog_plus := #JOG_PLUS_MODE AND NOT #JOG_MINUS_MODE AND NOT #REF_TRAVEL_MODE AND NOT #AUTO_OPTIMIZED AND NOT #AUTO_CW AND NOT #AUTO_CCW AND NOT #AUTO_PULS_MODE_CW AND NOT #AUTO_PULS_MODE_CCW;
END_REGION

REGION Network 16: Definition of modes: Jog minus selected
   #PO.Jog_minus := NOT #JOG_PLUS_MODE AND #JOG_MINUS_MODE AND NOT #REF_TRAVEL_MODE AND NOT #AUTO_OPTIMIZED AND NOT #AUTO_CW AND NOT #AUTO_CCW AND NOT #AUTO_PULS_MODE_CW AND NOT #AUTO_PULS_MODE_CCW;
END_REGION

REGION Network 17: Definition of modes: Ref selected
   #tRef := NOT #JOG_PLUS_MODE AND NOT #JOG_MINUS_MODE AND #REF_TRAVEL_MODE AND NOT #AUTO_OPTIMIZED AND NOT #AUTO_CW AND NOT #AUTO_CCW AND NOT #AUTO_PULS_MODE_CW AND NOT #AUTO_PULS_MODE_CCW;
END_REGION

REGION Network 18: Definition of modes: Auto opt.
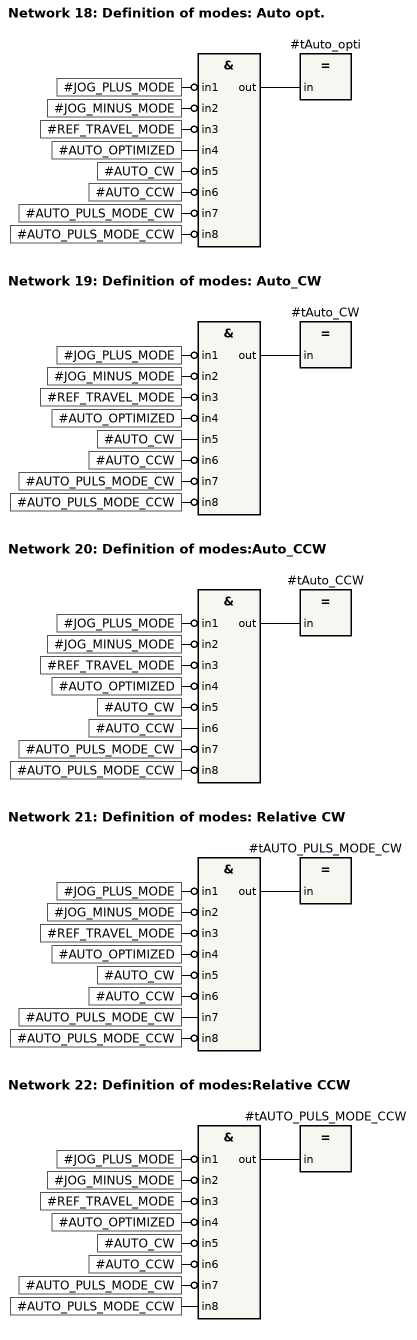
   #tAuto_opti := NOT #JOG_PLUS_MODE AND NOT #JOG_MINUS_MODE AND NOT #REF_TRAVEL_MODE AND #AUTO_OPTIMIZED AND NOT #AUTO_CW AND NOT #AUTO_CCW AND NOT #AUTO_PULS_MODE_CW AND NOT #AUTO_PULS_MODE_CCW;
END_REGION

REGION Network 19: Definition of modes: Auto_CW
   #tAuto_CW := NOT #JOG_PLUS_MODE AND NOT #JOG_MINUS_MODE AND NOT #REF_TRAVEL_MODE AND NOT #AUTO_OPTIMIZED AND #AUTO_CW AND NOT #AUTO_CCW AND NOT #AUTO_PULS_MODE_CW AND NOT #AUTO_PULS_MODE_CCW;
END_REGION

REGION Network 20: Definition of modes:Auto_CCW
   #tAuto_CCW := NOT #JOG_PLUS_MODE AND NOT #JOG_MINUS_MODE AND NOT #REF_TRAVEL_MODE AND NOT #AUTO_OPTIMIZED AND NOT #AUTO_CW AND #AUTO_CCW AND NOT #AUTO_PULS_MODE_CW AND NOT #AUTO_PULS_MODE_CCW;
END_REGION

REGION Network 21: Definition of modes: Relative CW
   #tAUTO_PULS_MODE_CW := NOT #JOG_PLUS_MODE AND NOT #JOG_MINUS_MODE AND NOT #REF_TRAVEL_MODE AND NOT #AUTO_OPTIMIZED AND NOT #AUTO_CW AND NOT #AUTO_CCW AND #AUTO_PULS_MODE_CW AND NOT #AUTO_PULS_MODE_CCW;
END_REGION

REGION Network 22: Definition of modes:Relative CCW
   #tAUTO_PULS_MODE_CCW := NOT #JOG_PLUS_MODE AND NOT #JOG_MINUS_MODE AND NOT #REF_TRAVEL_MODE AND NOT #AUTO_OPTIMIZED AND NOT #AUTO_CW AND NOT #AUTO_CCW AND NOT #AUTO_PULS_MODE_CW AND #AUTO_PULS_MODE_CCW;
END_REGION

REGION Network 23: Definition of modes: Bit11; / Definition der Modi: Anwahl "mode_low"
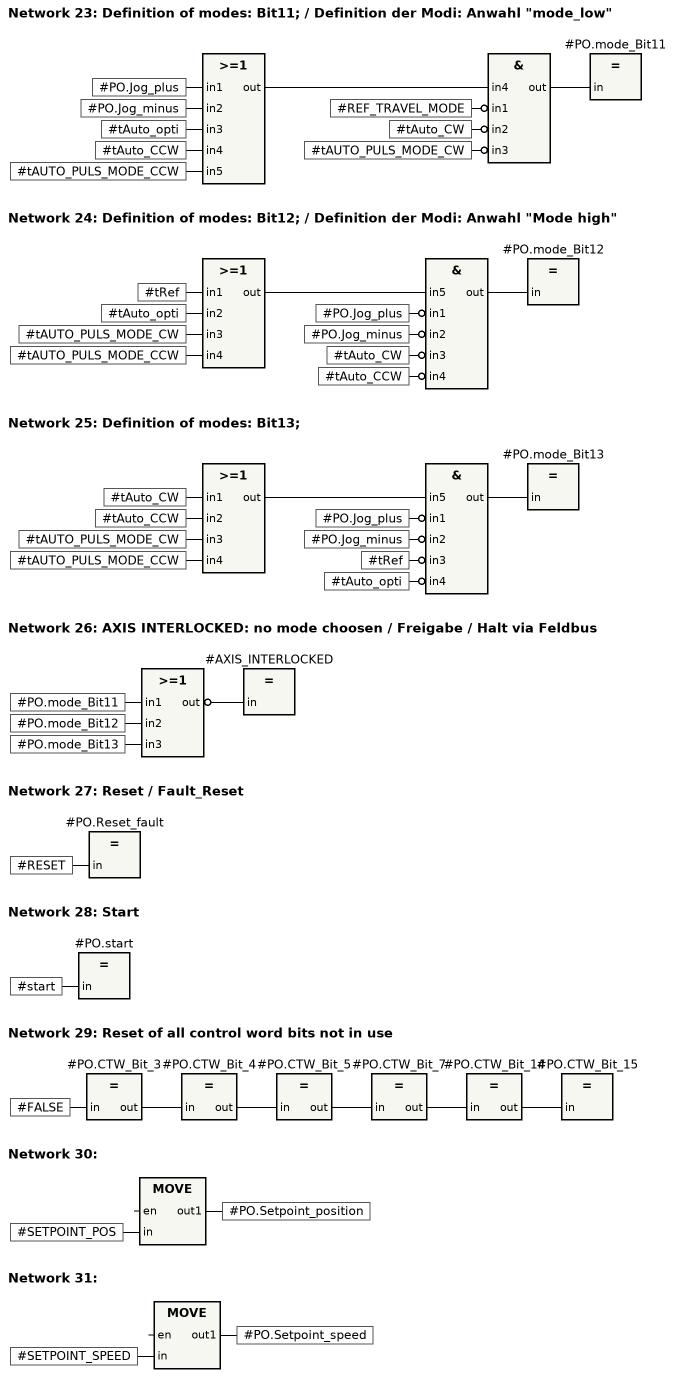
   #PO.mode_Bit11 := (#PO.Jog_plus OR #PO.Jog_minus OR #tAuto_opti OR #tAuto_CCW OR #tAUTO_PULS_MODE_CCW) AND NOT #REF_TRAVEL_MODE AND NOT #tAuto_CW AND NOT #tAUTO_PULS_MODE_CW;
END_REGION

REGION Network 24: Definition of modes: Bit12; / Definition der Modi: Anwahl "Mode high"
   #PO.mode_Bit12 := (#tRef OR #tAuto_opti OR #tAUTO_PULS_MODE_CW OR #tAUTO_PULS_MODE_CCW) AND NOT #PO.Jog_plus AND NOT #PO.Jog_minus AND NOT #tAuto_CW AND NOT #tAuto_CCW;
END_REGION

REGION Network 25: Definition of modes: Bit13;
   #PO.mode_Bit13 := (#tAuto_CW OR #tAuto_CCW OR #tAUTO_PULS_MODE_CW OR #tAUTO_PULS_MODE_CCW) AND NOT #PO.Jog_plus AND NOT #PO.Jog_minus AND NOT #tRef AND NOT #tAuto_opti;
END_REGION

REGION Network 26: AXIS INTERLOCKED: no mode choosen / Freigabe / Halt via Feldbus
   #AXIS_INTERLOCKED := NOT (#PO.mode_Bit11 OR #PO.mode_Bit12 OR #PO.mode_Bit13);
END_REGION

REGION Network 27: Reset / Fault_Reset
   #PO.Reset_fault := #RESET;
END_REGION

REGION Network 28: Start
   #PO.start := #start;
END_REGION

REGION Network 29: Reset of all control word bits not in use
   #PO.CTW_Bit_3 := #FALSE;
   #PO.CTW_Bit_4 := #FALSE;
   #PO.CTW_Bit_5 := #FALSE;
   #PO.CTW_Bit_7 := #FALSE;
   #PO.CTW_Bit_14 := #FALSE;
   #PO.CTW_Bit_15 := #FALSE;
END_REGION

REGION Network 30
   #PO.Setpoint_position := #SETPOINT_POS;
END_REGION

REGION Network 31
   #PO.Setpoint_speed := #SETPOINT_SPEED;
END_REGION

REGION Network 32: Start/Stop-ramp
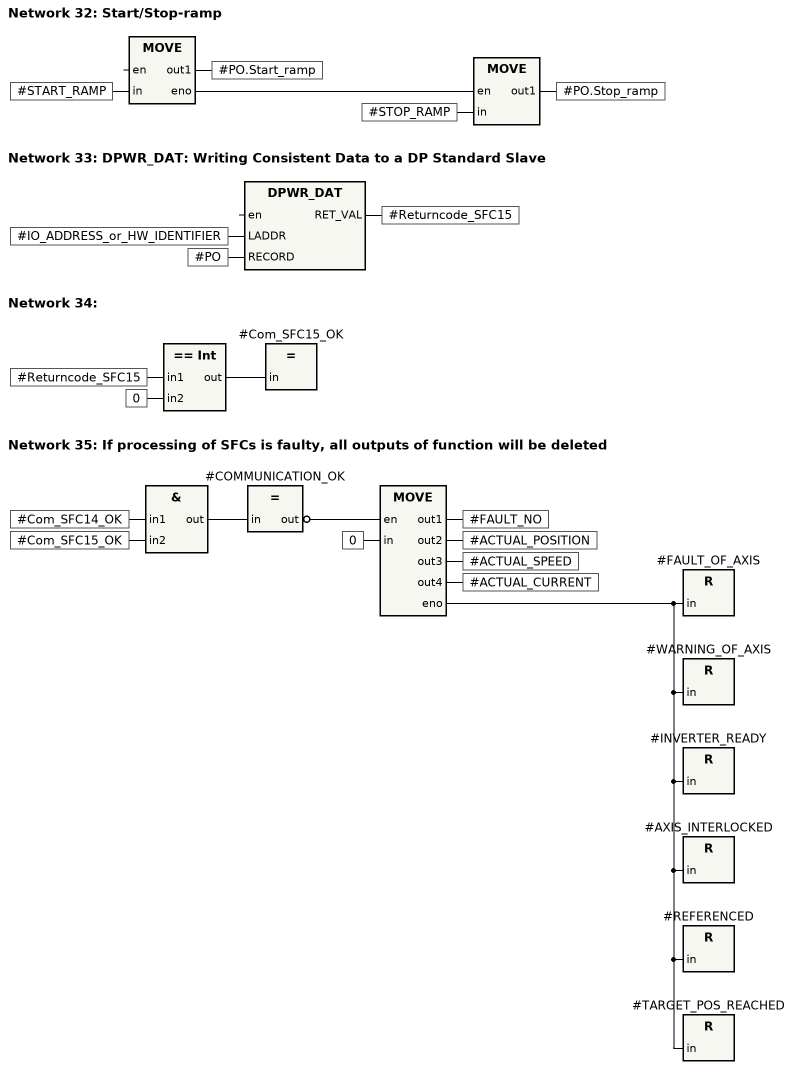
   // ENO of a box is taken as its EN; it also drops when the box reports an error
   #PO.Start_ramp := #START_RAMP;
   #PO.Stop_ramp := #STOP_RAMP;
END_REGION

REGION Network 33: DPWR_DAT: Writing Consistent Data to a DP Standard Slave
   #Returncode_SFC15 := DPWR_DAT(LADDR := #IO_ADDRESS_or_HW_IDENTIFIER, RECORD := #PO);
END_REGION

REGION Network 34
   #Com_SFC15_OK := #Returncode_SFC15 = 0;
END_REGION

REGION Network 35: If processing of SFCs is faulty, all outputs of function will be deleted
   // ENO of a box is taken as its EN; it also drops when the box reports an error
   END:
   #_w1 := #Com_SFC14_OK AND #Com_SFC15_OK;
   #COMMUNICATION_OK := #_w1;
   IF NOT #_w1 THEN
       #FAULT_NO := 0;
       #ACTUAL_POSITION := 0;
       #ACTUAL_SPEED := 0;
       #ACTUAL_CURRENT := 0;
       #FAULT_OF_AXIS := FALSE;
       #WARNING_OF_AXIS := FALSE;
       #INVERTER_READY := FALSE;
       #AXIS_INTERLOCKED := FALSE;
       #REFERENCED := FALSE;
       #TARGET_POS_REACHED := FALSE;
   END_IF;
END_REGION
END_FUNCTION

ORGANIZATION_BLOCK "Main"   // OB1, LAD, ProgramCycle
TITLE = "Main Program Sweep (Cycle)"
{ S7_Optimized_Access := 'TRUE' }
VERSION : 0.1
   VAR_INPUT
      Initial_Call : Bool;   // Initial call of this OB
      Remanence : Bool;   // =True, if remanent data are available
   END_VAR
   VAR CONSTANT
      Aviso1 : Time := T#4s;
      Aviso2 : Time := T#7ms;
      Aviso_Giro : Time := T#10s;
   END_VAR
   VAR_TEMP   // added for the SCL form of the ladder/FBD networks
      _w1 : Bool;
      _w2 : Bool;
   END_VAR
BEGIN

REGION Network 1: SEMPRE 0
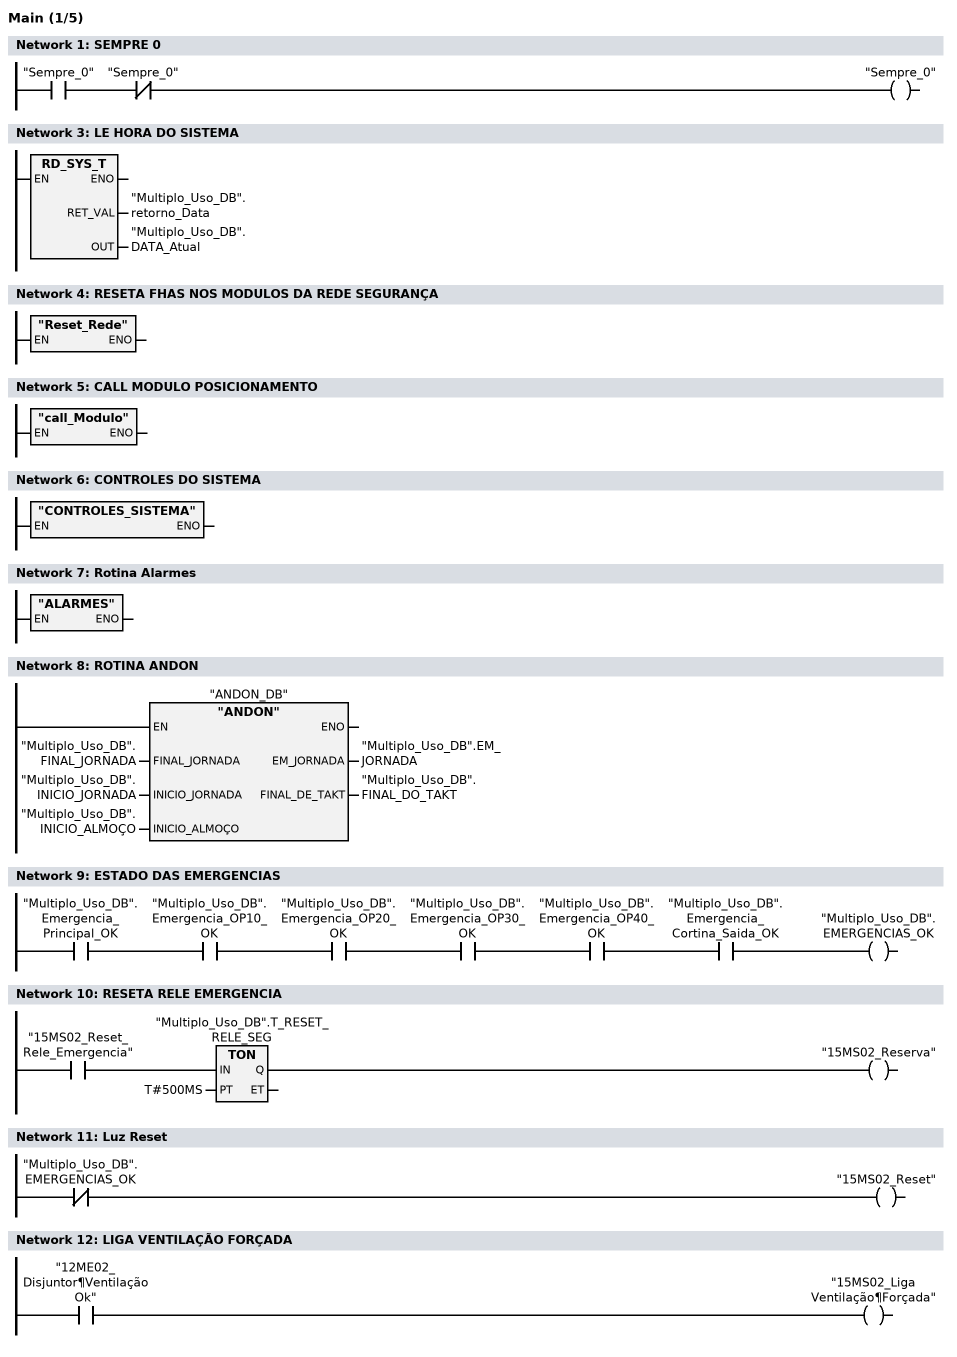
   RUNG wire#powerrail
      Contact( "Sempre_0" )
      I_Contact( "Sempre_0" )
      Coil( "Sempre_0" )
   END_RUNG
   // the same network as SCL:
   "Sempre_0" := "Sempre_0" AND NOT "Sempre_0";
END_REGION

REGION Network 3: LE HORA DO SISTEMA
   "Multiplo_Uso_DB".retorno_Data := RD_SYS_T(OUT => "Multiplo_Uso_DB".DATA_Atual);
END_REGION

REGION Network 4: RESETA FHAS NOS MODULOS DA REDE SEGURANÇA
   RUNG wire#powerrail
      "Reset_Rede"()
   END_RUNG
   // the same network as SCL:
   "Reset_Rede"();
END_REGION

REGION Network 5: CALL MODULO POSICIONAMENTO
   RUNG wire#powerrail
      "call_Modulo"()
   END_RUNG
   // the same network as SCL:
   "call_Modulo"();
END_REGION

REGION Network 6: CONTROLES DO SISTEMA
   RUNG wire#powerrail
      "CONTROLES_SISTEMA"()
   END_RUNG
   // the same network as SCL:
   "CONTROLES_SISTEMA"();
END_REGION

REGION Network 7: Rotina Alarmes
   RUNG wire#powerrail
      "ALARMES"()
   END_RUNG
   // the same network as SCL:
   "ALARMES"();
END_REGION

REGION Network 8: ROTINA ANDON
   RUNG wire#powerrail
      "ANDON_DB"(FINAL_JORNADA := "Multiplo_Uso_DB".FINAL_JORNADA, INICIO_JORNADA := "Multiplo_Uso_DB".INICIO_JORNADA, INICIO_ALMOÇO := "Multiplo_Uso_DB".INICIO_ALMOÇO, EM_JORNADA => "Multiplo_Uso_DB".EM_JORNADA, FINAL_DE_TAKT => "Multiplo_Uso_DB".FINAL_DO_TAKT)
   END_RUNG
   // the same network as SCL:
   "ANDON_DB"(FINAL_JORNADA := "Multiplo_Uso_DB".FINAL_JORNADA,   // "ANDON"
              INICIO_JORNADA := "Multiplo_Uso_DB".INICIO_JORNADA,
              INICIO_ALMOÇO := "Multiplo_Uso_DB".INICIO_ALMOÇO,
              EM_JORNADA => "Multiplo_Uso_DB".EM_JORNADA,
              FINAL_DE_TAKT => "Multiplo_Uso_DB".FINAL_DO_TAKT);
END_REGION

REGION Network 9: ESTADO DAS EMERGENCIAS
   RUNG wire#powerrail
      Contact( "Multiplo_Uso_DB".Emergencia_Principal_OK )
      Contact( "Multiplo_Uso_DB".Emergencia_OP10_OK )
      Contact( "Multiplo_Uso_DB".Emergencia_OP20_OK )
      Contact( "Multiplo_Uso_DB".Emergencia_OP30_OK )
      Contact( "Multiplo_Uso_DB".Emergencia_OP40_OK )
      Contact( "Multiplo_Uso_DB".Emergencia_Cortina_Saida_OK )
      Coil( "Multiplo_Uso_DB".EMERGENCIAS_OK )
   END_RUNG
   // the same network as SCL:
   "Multiplo_Uso_DB".EMERGENCIAS_OK := "Multiplo_Uso_DB".Emergencia_Principal_OK AND "Multiplo_Uso_DB".Emergencia_OP10_OK AND "Multiplo_Uso_DB".Emergencia_OP20_OK AND "Multiplo_Uso_DB".Emergencia_OP30_OK AND "Multiplo_Uso_DB".Emergencia_OP40_OK AND "Multiplo_Uso_DB".Emergencia_Cortina_Saida_OK;
END_REGION

REGION Network 10: RESETA RELE EMERGENCIA
   "Multiplo_Uso_DB".T_RESET_RELE_SEG.TON(IN := "15MS02_Reset_Rele_Emergencia", PT := T#500MS);
   "15MS02_Reserva" := "Multiplo_Uso_DB".T_RESET_RELE_SEG.Q;
END_REGION

REGION Network 11: Luz Reset
   RUNG wire#powerrail
      I_Contact( "Multiplo_Uso_DB".EMERGENCIAS_OK )
      Coil( "15MS02_Reset" )
   END_RUNG
   // the same network as SCL:
   "15MS02_Reset" := NOT "Multiplo_Uso_DB".EMERGENCIAS_OK;
END_REGION

REGION Network 12: LIGA VENTILAÇÃO FORÇADA
   RUNG wire#powerrail
      Contact( "12ME02_Disjuntor¶Ventilação Ok" )
      Coil( "15MS02_Liga Ventilação¶Forçada" )
   END_RUNG
   // the same network as SCL:
   "15MS02_Liga Ventilação¶Forçada" := "12ME02_Disjuntor¶Ventilação Ok";
END_REGION

REGION Network 13: VERIFICA TODAS OPERAÇÕES OK
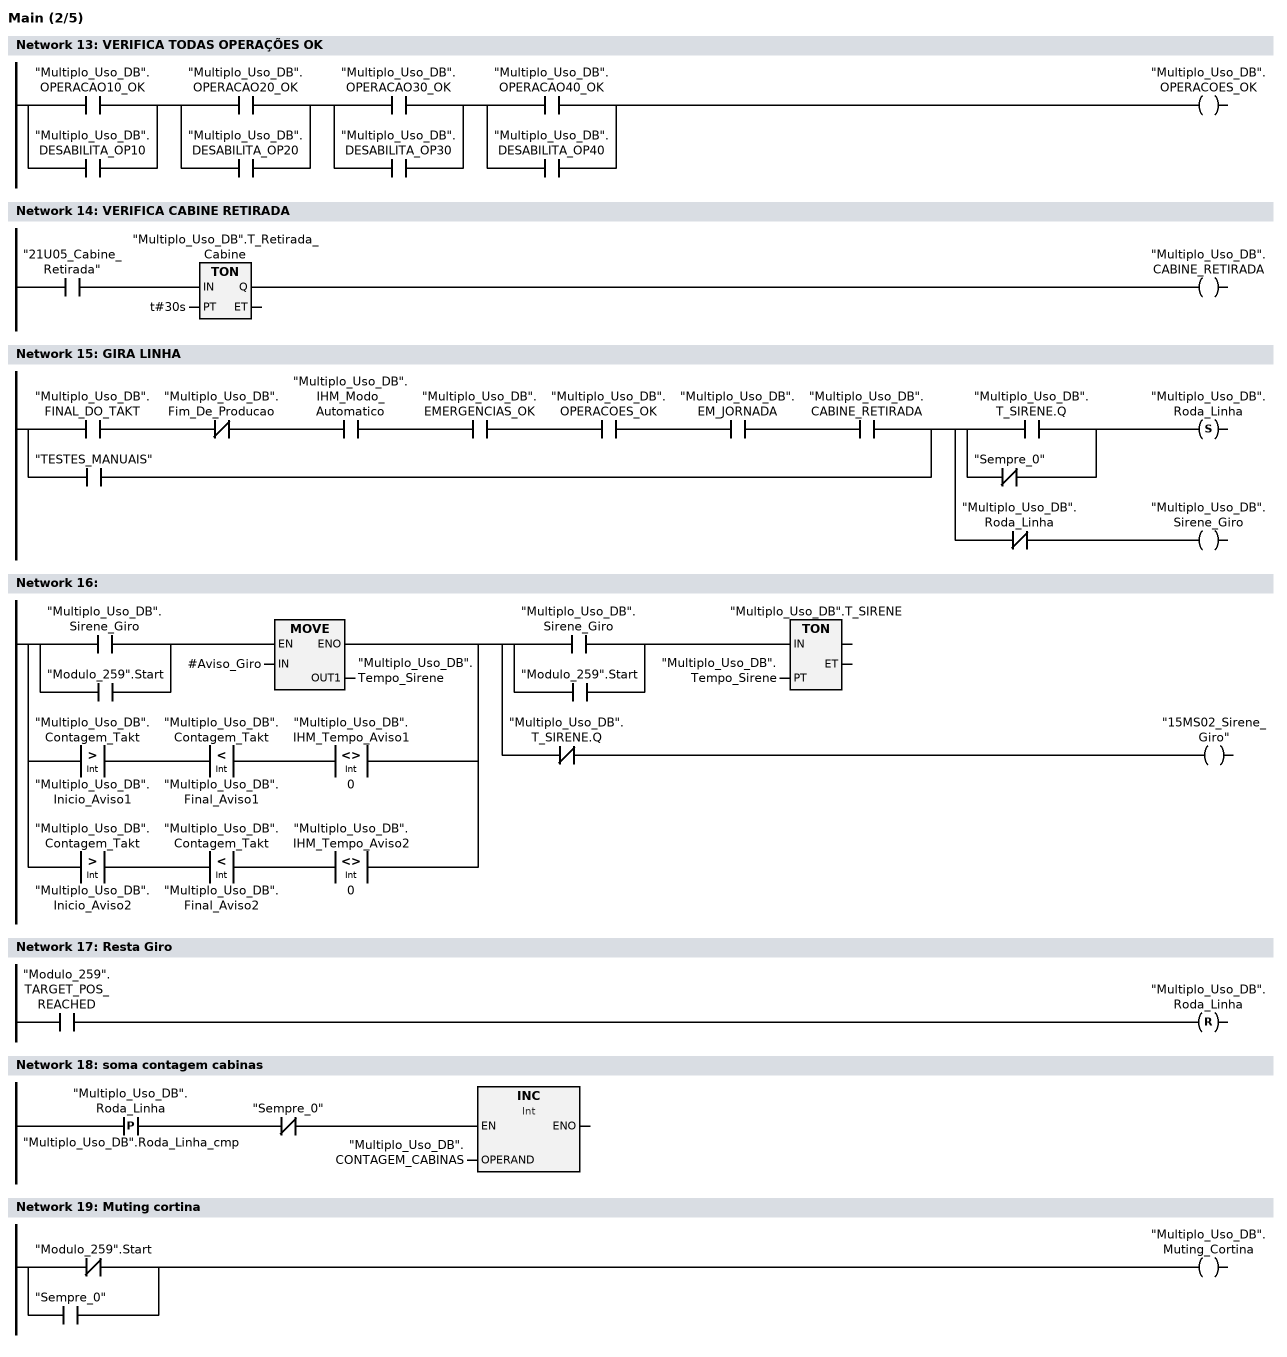
   RUNG wire#powerrail
      Contact( "Multiplo_Uso_DB".OPERACAO10_OK )
      wire#w1
      Contact( "Multiplo_Uso_DB".OPERACAO20_OK )
      wire#w2
      Contact( "Multiplo_Uso_DB".OPERACAO30_OK )
      wire#w3
      Contact( "Multiplo_Uso_DB".OPERACAO40_OK )
      wire#w4
      Coil( "Multiplo_Uso_DB".OPERACOES_OK )
   END_RUNG
   RUNG wire#powerrail
      Contact( "Multiplo_Uso_DB".DESABILITA_OP10 )
   END_RUNG wire#w1
   RUNG wire#w1
      Contact( "Multiplo_Uso_DB".DESABILITA_OP20 )
   END_RUNG wire#w2
   RUNG wire#w2
      Contact( "Multiplo_Uso_DB".DESABILITA_OP30 )
   END_RUNG wire#w3
   RUNG wire#w3
      Contact( "Multiplo_Uso_DB".DESABILITA_OP40 )
   END_RUNG wire#w4
   // the same network as SCL:
   "Multiplo_Uso_DB".OPERACOES_OK := ("Multiplo_Uso_DB".OPERACAO10_OK OR "Multiplo_Uso_DB".DESABILITA_OP10) AND ("Multiplo_Uso_DB".OPERACAO20_OK OR "Multiplo_Uso_DB".DESABILITA_OP20) AND ("Multiplo_Uso_DB".OPERACAO30_OK OR "Multiplo_Uso_DB".DESABILITA_OP30) AND ("Multiplo_Uso_DB".OPERACAO40_OK OR "Multiplo_Uso_DB".DESABILITA_OP40);
END_REGION

REGION Network 14: VERIFICA CABINE RETIRADA
   "Multiplo_Uso_DB".T_Retirada_Cabine.TON(IN := "21U05_Cabine_Retirada", PT := t#30s);
   "Multiplo_Uso_DB".CABINE_RETIRADA := "Multiplo_Uso_DB".T_Retirada_Cabine.Q;
END_REGION

REGION Network 15: GIRA LINHA
   RUNG wire#powerrail
      Contact( "Multiplo_Uso_DB".FINAL_DO_TAKT )
      I_Contact( "Multiplo_Uso_DB".Fim_De_Producao )
      Contact( "Multiplo_Uso_DB".IHM_Modo_Automatico )
      Contact( "Multiplo_Uso_DB".EMERGENCIAS_OK )
      Contact( "Multiplo_Uso_DB".OPERACOES_OK )
      Contact( "Multiplo_Uso_DB".EM_JORNADA )
      Contact( "Multiplo_Uso_DB".CABINE_RETIRADA )
      wire#w1
      Contact( "Multiplo_Uso_DB".T_SIRENE.Q )
      wire#w2
      S_Coil( "Multiplo_Uso_DB".Roda_Linha )
   END_RUNG
   RUNG wire#powerrail
      Contact( "TESTES_MANUAIS" )
   END_RUNG wire#w1
   RUNG wire#w1
      I_Contact( "Sempre_0" )
   END_RUNG wire#w2
   RUNG wire#w1
      I_Contact( "Multiplo_Uso_DB".Roda_Linha )
      Coil( "Multiplo_Uso_DB".Sirene_Giro )
   END_RUNG
   // the same network as SCL:
   #_w1 := ("Multiplo_Uso_DB".FINAL_DO_TAKT AND NOT "Multiplo_Uso_DB".Fim_De_Producao AND "Multiplo_Uso_DB".IHM_Modo_Automatico AND "Multiplo_Uso_DB".EMERGENCIAS_OK AND "Multiplo_Uso_DB".OPERACOES_OK AND "Multiplo_Uso_DB".EM_JORNADA AND "Multiplo_Uso_DB".CABINE_RETIRADA) OR "TESTES_MANUAIS";
   IF #_w1 AND ("Multiplo_Uso_DB".T_SIRENE.Q OR NOT "Sempre_0") THEN
       "Multiplo_Uso_DB".Roda_Linha := TRUE;
   END_IF;
   "Multiplo_Uso_DB".Sirene_Giro := #_w1 AND NOT "Multiplo_Uso_DB".Roda_Linha;
END_REGION

REGION Network 16
   #_w1 := "Multiplo_Uso_DB".Sirene_Giro OR "Modulo_259".Start;
   IF #_w1 THEN "Multiplo_Uso_DB".Tempo_Sirene := #Aviso_Giro; END_IF;
   #_w2 := #_w1 OR (("Multiplo_Uso_DB".Contagem_Takt > "Multiplo_Uso_DB".Inicio_Aviso1) AND ("Multiplo_Uso_DB".Contagem_Takt < "Multiplo_Uso_DB".Final_Aviso1) AND ("Multiplo_Uso_DB".IHM_Tempo_Aviso1 <> 0)) OR (("Multiplo_Uso_DB".Contagem_Takt > "Multiplo_Uso_DB".Inicio_Aviso2) AND ("Multiplo_Uso_DB".Contagem_Takt < "Multiplo_Uso_DB".Final_Aviso2) AND ("Multiplo_Uso_DB".IHM_Tempo_Aviso2 <> 0));
   "Multiplo_Uso_DB".T_SIRENE.TON(IN := #_w2 AND ("Multiplo_Uso_DB".Sirene_Giro OR "Modulo_259".Start),
                           PT := "Multiplo_Uso_DB".Tempo_Sirene);
   "15MS02_Sirene_Giro" := #_w2 AND NOT "Multiplo_Uso_DB".T_SIRENE.Q;
END_REGION

REGION Network 17: Resta Giro
   RUNG wire#powerrail
      Contact( "Modulo_259".TARGET_POS_REACHED )
      R_Coil( "Multiplo_Uso_DB".Roda_Linha )
   END_RUNG
   // the same network as SCL:
   IF "Modulo_259".TARGET_POS_REACHED THEN "Multiplo_Uso_DB".Roda_Linha := FALSE; END_IF;
END_REGION

REGION Network 18: soma contagem cabinas
   RUNG wire#powerrail
      P_Contact(operand := "Multiplo_Uso_DB".Roda_Linha, bit := "Multiplo_Uso_DB".Roda_Linha_cmp)
      I_Contact( "Sempre_0" )
      { S7_Templates := "DestType := Int" } Inc( "Multiplo_Uso_DB".CONTAGEM_CABINAS )
   END_RUNG
   // the same network as SCL:
   #_w1 := "Multiplo_Uso_DB".Roda_Linha AND NOT "Multiplo_Uso_DB".Roda_Linha_cmp;   // rising edge of "Multiplo_Uso_DB".Roda_Linha
   "Multiplo_Uso_DB".Roda_Linha_cmp := "Multiplo_Uso_DB".Roda_Linha;
   IF #_w1 AND NOT "Sempre_0" THEN
       "Multiplo_Uso_DB".CONTAGEM_CABINAS := "Multiplo_Uso_DB".CONTAGEM_CABINAS + 1;
   END_IF;
END_REGION

REGION Network 19: Muting cortina
   RUNG wire#powerrail
      I_Contact( "Modulo_259".Start )
      wire#w1
      Coil( "Multiplo_Uso_DB".Muting_Cortina )
   END_RUNG
   RUNG wire#powerrail
      Contact( "Sempre_0" )
   END_RUNG wire#w1
   // the same network as SCL:
   "Multiplo_Uso_DB".Muting_Cortina := NOT "Modulo_259".Start OR "Sempre_0";
END_REGION

REGION Network 20: Habilita Muting
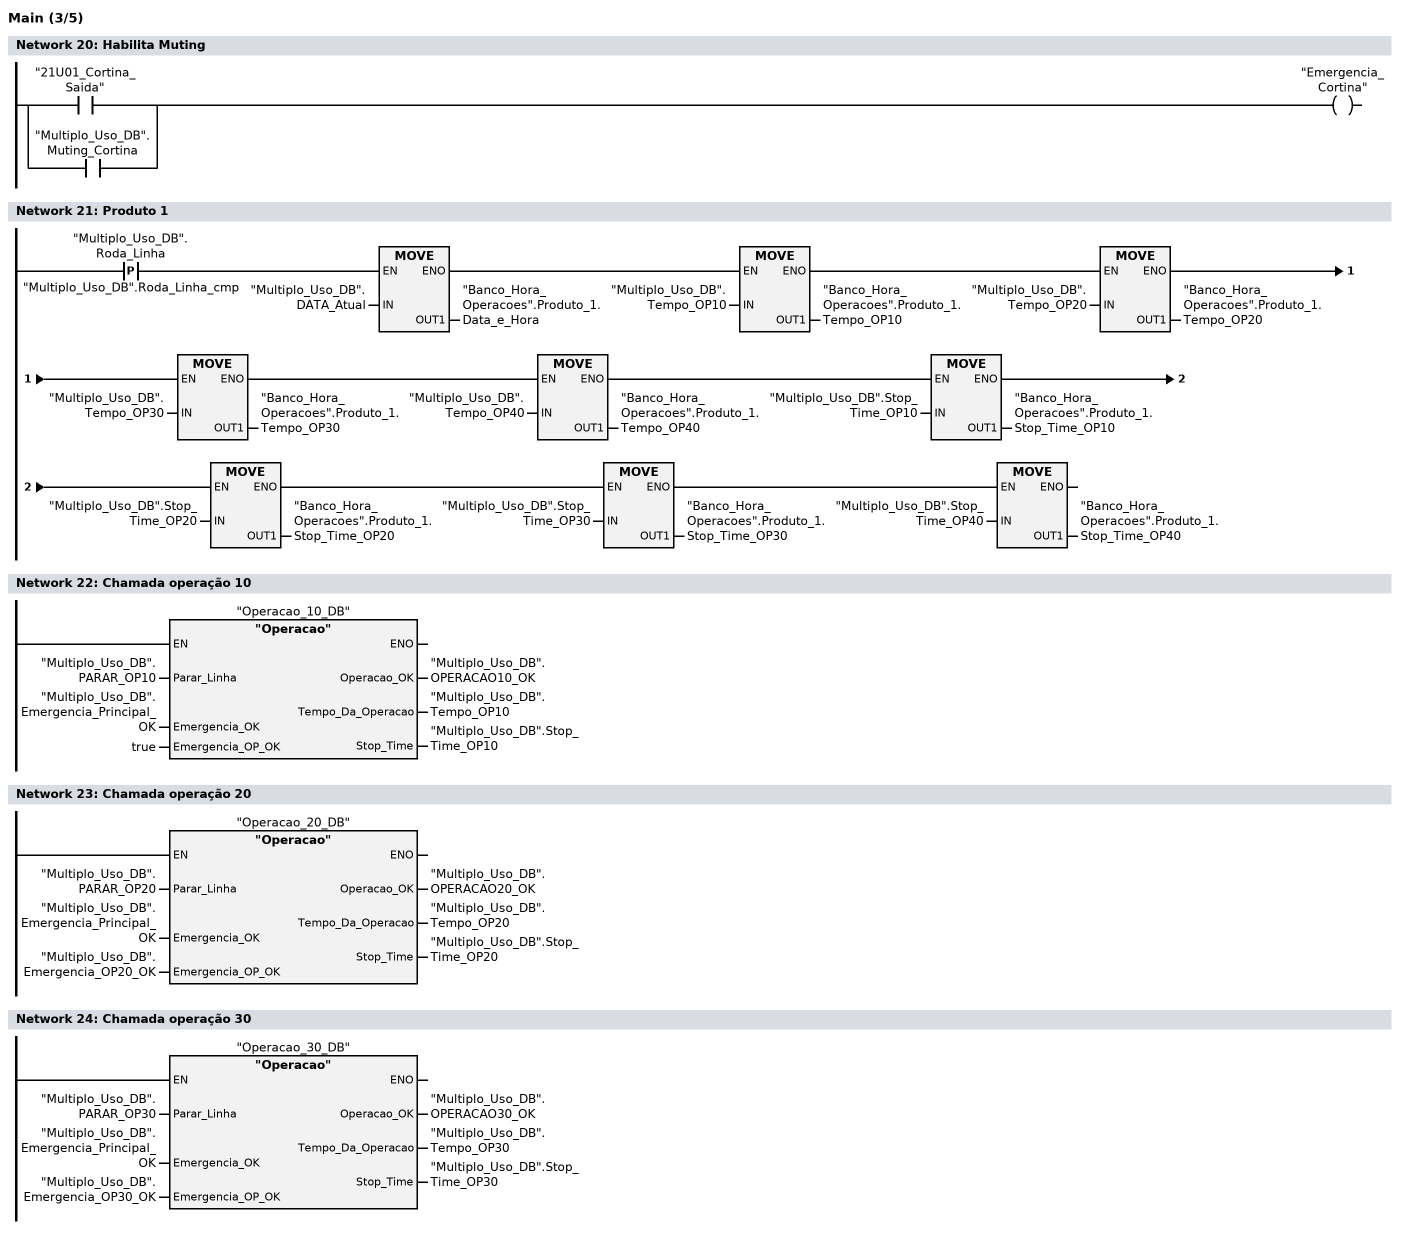
   RUNG wire#powerrail
      Contact( "21U01_Cortina_Saida" )
      wire#w1
      Coil( "Emergencia_Cortina" )
   END_RUNG
   RUNG wire#powerrail
      Contact( "Multiplo_Uso_DB".Muting_Cortina )
   END_RUNG wire#w1
   // the same network as SCL:
   "Emergencia_Cortina" := "21U01_Cortina_Saida" OR "Multiplo_Uso_DB".Muting_Cortina;
END_REGION

REGION Network 21: Produto 1
   RUNG wire#powerrail
      P_Contact(operand := "Multiplo_Uso_DB".Roda_Linha, bit := "Multiplo_Uso_DB".Roda_Linha_cmp)
      Move(in := "Multiplo_Uso_DB".DATA_Atual, out1 => "Banco_Hora_Operacoes".Produto_1.Data_e_Hora)
      Move(in := "Multiplo_Uso_DB".Tempo_OP10, out1 => "Banco_Hora_Operacoes".Produto_1.Tempo_OP10)
      Move(in := "Multiplo_Uso_DB".Tempo_OP20, out1 => "Banco_Hora_Operacoes".Produto_1.Tempo_OP20)
      Move(in := "Multiplo_Uso_DB".Tempo_OP30, out1 => "Banco_Hora_Operacoes".Produto_1.Tempo_OP30)
      Move(in := "Multiplo_Uso_DB".Tempo_OP40, out1 => "Banco_Hora_Operacoes".Produto_1.Tempo_OP40)
      Move(in := "Multiplo_Uso_DB".Stop_Time_OP10, out1 => "Banco_Hora_Operacoes".Produto_1.Stop_Time_OP10)
      Move(in := "Multiplo_Uso_DB".Stop_Time_OP20, out1 => "Banco_Hora_Operacoes".Produto_1.Stop_Time_OP20)
      Move(in := "Multiplo_Uso_DB".Stop_Time_OP30, out1 => "Banco_Hora_Operacoes".Produto_1.Stop_Time_OP30)
      Move(in := "Multiplo_Uso_DB".Stop_Time_OP40, out1 => "Banco_Hora_Operacoes".Produto_1.Stop_Time_OP40)
   END_RUNG
   // the same network as SCL:
   #_w1 := "Multiplo_Uso_DB".Roda_Linha AND NOT "Multiplo_Uso_DB".Roda_Linha_cmp;   // rising edge of "Multiplo_Uso_DB".Roda_Linha
   "Multiplo_Uso_DB".Roda_Linha_cmp := "Multiplo_Uso_DB".Roda_Linha;
   IF #_w1 THEN
       "Banco_Hora_Operacoes".Produto_1.Data_e_Hora := "Multiplo_Uso_DB".DATA_Atual;
       "Banco_Hora_Operacoes".Produto_1.Tempo_OP10 := "Multiplo_Uso_DB".Tempo_OP10;
       "Banco_Hora_Operacoes".Produto_1.Tempo_OP20 := "Multiplo_Uso_DB".Tempo_OP20;
       "Banco_Hora_Operacoes".Produto_1.Tempo_OP30 := "Multiplo_Uso_DB".Tempo_OP30;
       "Banco_Hora_Operacoes".Produto_1.Tempo_OP40 := "Multiplo_Uso_DB".Tempo_OP40;
       "Banco_Hora_Operacoes".Produto_1.Stop_Time_OP10 := "Multiplo_Uso_DB".Stop_Time_OP10;
       "Banco_Hora_Operacoes".Produto_1.Stop_Time_OP20 := "Multiplo_Uso_DB".Stop_Time_OP20;
       "Banco_Hora_Operacoes".Produto_1.Stop_Time_OP30 := "Multiplo_Uso_DB".Stop_Time_OP30;
       "Banco_Hora_Operacoes".Produto_1.Stop_Time_OP40 := "Multiplo_Uso_DB".Stop_Time_OP40;
   END_IF;
END_REGION

REGION Network 22: Chamada operação 10
   RUNG wire#powerrail
      "Operacao_10_DB"(Parar_Linha := "Multiplo_Uso_DB".PARAR_OP10, Emergencia_OK := "Multiplo_Uso_DB".Emergencia_Principal_OK, Emergencia_OP_OK := true, Operacao_OK => "Multiplo_Uso_DB".OPERACAO10_OK, Tempo_Da_Operacao => "Multiplo_Uso_DB".Tempo_OP10, Stop_Time => "Multiplo_Uso_DB".Stop_Time_OP10)
   END_RUNG
   // the same network as SCL:
   "Operacao_10_DB"(Parar_Linha := "Multiplo_Uso_DB".PARAR_OP10,   // "Operacao"
                    Emergencia_OK := "Multiplo_Uso_DB".Emergencia_Principal_OK,
                    Emergencia_OP_OK := true,
                    Operacao_OK => "Multiplo_Uso_DB".OPERACAO10_OK,
                    Tempo_Da_Operacao => "Multiplo_Uso_DB".Tempo_OP10,
                    Stop_Time => "Multiplo_Uso_DB".Stop_Time_OP10);
END_REGION

REGION Network 23: Chamada operação 20
   RUNG wire#powerrail
      "Operacao_20_DB"(Parar_Linha := "Multiplo_Uso_DB".PARAR_OP20, Emergencia_OK := "Multiplo_Uso_DB".Emergencia_Principal_OK, Emergencia_OP_OK := "Multiplo_Uso_DB".Emergencia_OP20_OK, Operacao_OK => "Multiplo_Uso_DB".OPERACAO20_OK, Tempo_Da_Operacao => "Multiplo_Uso_DB".Tempo_OP20, Stop_Time => "Multiplo_Uso_DB".Stop_Time_OP20)
   END_RUNG
   // the same network as SCL:
   "Operacao_20_DB"(Parar_Linha := "Multiplo_Uso_DB".PARAR_OP20,   // "Operacao"
                    Emergencia_OK := "Multiplo_Uso_DB".Emergencia_Principal_OK,
                    Emergencia_OP_OK := "Multiplo_Uso_DB".Emergencia_OP20_OK,
                    Operacao_OK => "Multiplo_Uso_DB".OPERACAO20_OK,
                    Tempo_Da_Operacao => "Multiplo_Uso_DB".Tempo_OP20,
                    Stop_Time => "Multiplo_Uso_DB".Stop_Time_OP20);
END_REGION

REGION Network 24: Chamada operação 30
   RUNG wire#powerrail
      "Operacao_30_DB"(Parar_Linha := "Multiplo_Uso_DB".PARAR_OP30, Emergencia_OK := "Multiplo_Uso_DB".Emergencia_Principal_OK, Emergencia_OP_OK := "Multiplo_Uso_DB".Emergencia_OP30_OK, Operacao_OK => "Multiplo_Uso_DB".OPERACAO30_OK, Tempo_Da_Operacao => "Multiplo_Uso_DB".Tempo_OP30, Stop_Time => "Multiplo_Uso_DB".Stop_Time_OP30)
   END_RUNG
   // the same network as SCL:
   "Operacao_30_DB"(Parar_Linha := "Multiplo_Uso_DB".PARAR_OP30,   // "Operacao"
                    Emergencia_OK := "Multiplo_Uso_DB".Emergencia_Principal_OK,
                    Emergencia_OP_OK := "Multiplo_Uso_DB".Emergencia_OP30_OK,
                    Operacao_OK => "Multiplo_Uso_DB".OPERACAO30_OK,
                    Tempo_Da_Operacao => "Multiplo_Uso_DB".Tempo_OP30,
                    Stop_Time => "Multiplo_Uso_DB".Stop_Time_OP30);
END_REGION

REGION Network 25: Chamada operação 40
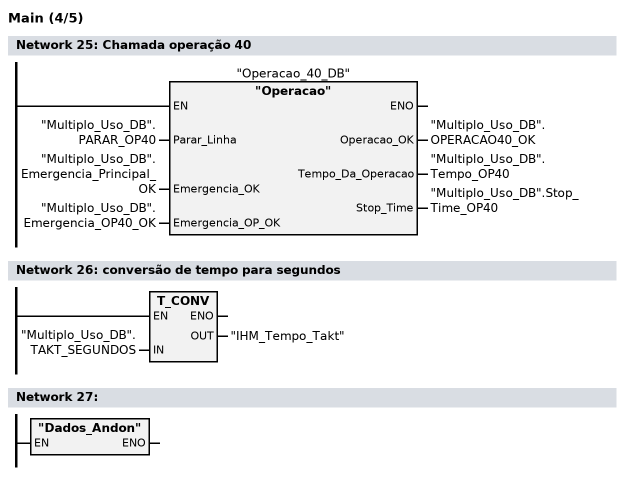
   RUNG wire#powerrail
      "Operacao_40_DB"(Parar_Linha := "Multiplo_Uso_DB".PARAR_OP40, Emergencia_OK := "Multiplo_Uso_DB".Emergencia_Principal_OK, Emergencia_OP_OK := "Multiplo_Uso_DB".Emergencia_OP40_OK, Operacao_OK => "Multiplo_Uso_DB".OPERACAO40_OK, Tempo_Da_Operacao => "Multiplo_Uso_DB".Tempo_OP40, Stop_Time => "Multiplo_Uso_DB".Stop_Time_OP40)
   END_RUNG
   // the same network as SCL:
   "Operacao_40_DB"(Parar_Linha := "Multiplo_Uso_DB".PARAR_OP40,   // "Operacao"
                    Emergencia_OK := "Multiplo_Uso_DB".Emergencia_Principal_OK,
                    Emergencia_OP_OK := "Multiplo_Uso_DB".Emergencia_OP40_OK,
                    Operacao_OK => "Multiplo_Uso_DB".OPERACAO40_OK,
                    Tempo_Da_Operacao => "Multiplo_Uso_DB".Tempo_OP40,
                    Stop_Time => "Multiplo_Uso_DB".Stop_Time_OP40);
END_REGION

REGION Network 26: conversão de tempo para segundos
   "IHM_Tempo_Takt" := T_CONV(IN := "Multiplo_Uso_DB".TAKT_SEGUNDOS);
END_REGION

REGION Network 27
   RUNG wire#powerrail
      "Dados_Andon"()
   END_RUNG
   // the same network as SCL:
   "Dados_Andon"();
END_REGION

REGION Network 29
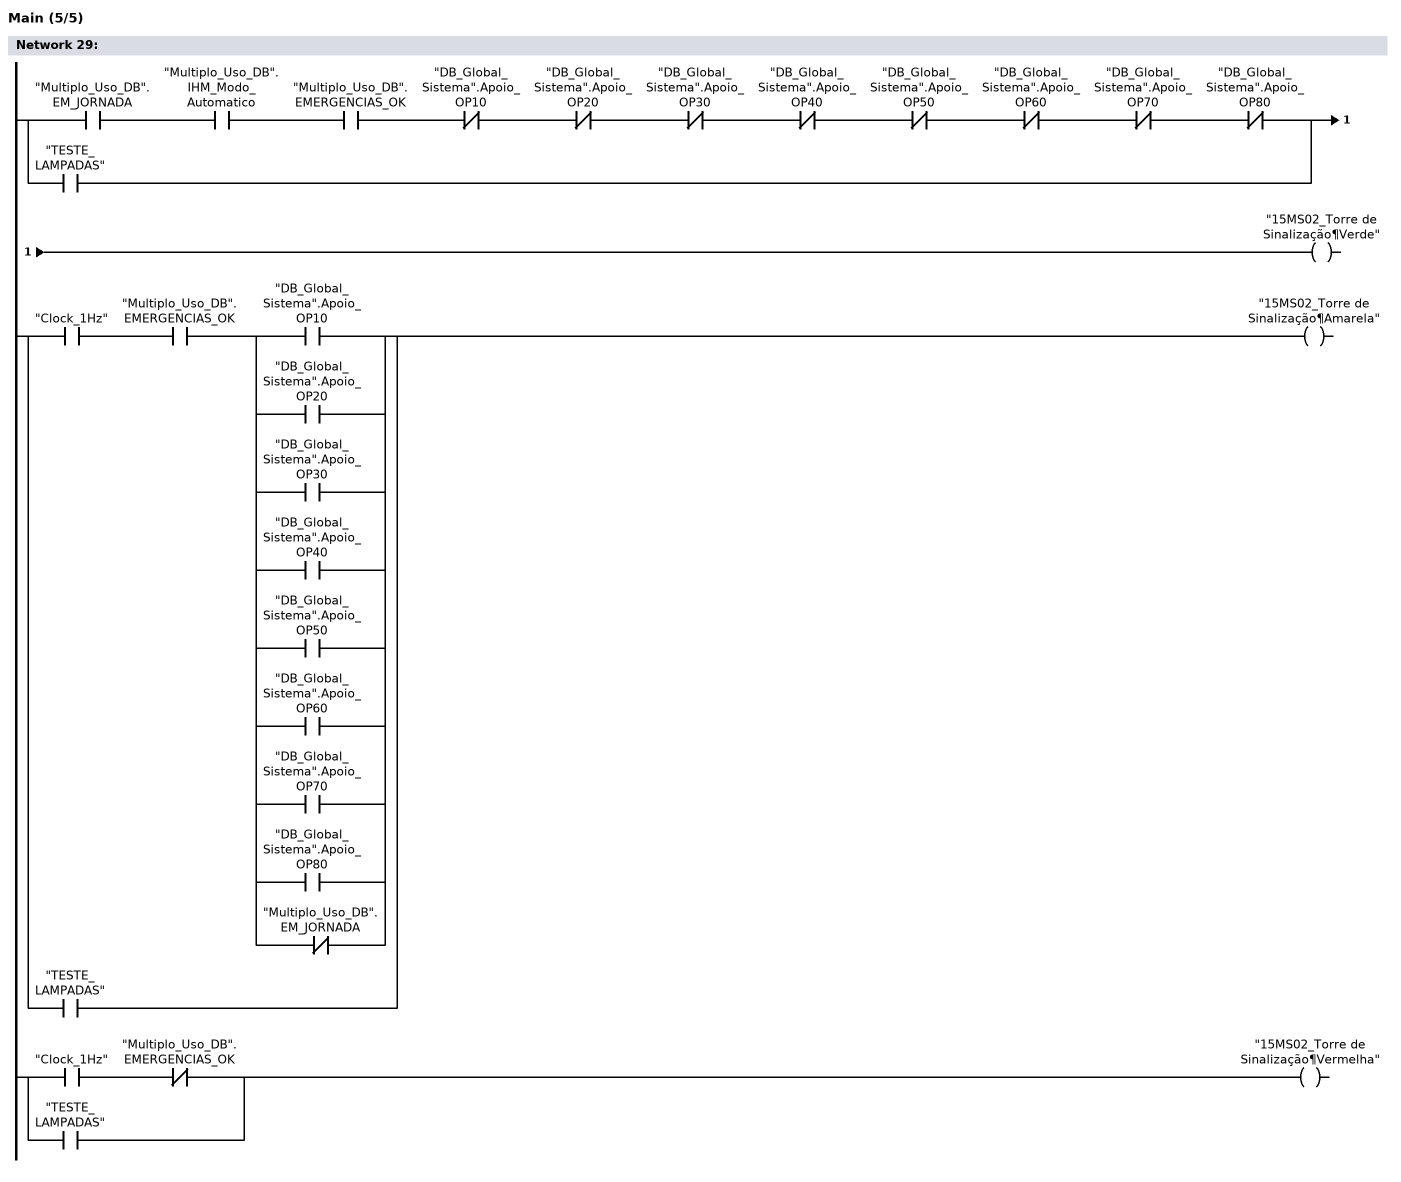
   RUNG wire#powerrail
      Contact( "Multiplo_Uso_DB".EM_JORNADA )
      Contact( "Multiplo_Uso_DB".IHM_Modo_Automatico )
      Contact( "Multiplo_Uso_DB".EMERGENCIAS_OK )
      I_Contact( "DB_Global_Sistema".Apoio_OP10 )
      I_Contact( "DB_Global_Sistema".Apoio_OP20 )
      I_Contact( "DB_Global_Sistema".Apoio_OP30 )
      I_Contact( "DB_Global_Sistema".Apoio_OP40 )
      I_Contact( "DB_Global_Sistema".Apoio_OP50 )
      I_Contact( "DB_Global_Sistema".Apoio_OP60 )
      I_Contact( "DB_Global_Sistema".Apoio_OP70 )
      I_Contact( "DB_Global_Sistema".Apoio_OP80 )
      wire#w1
      Coil( "15MS02_Torre de Sinalização¶Verde" )
   END_RUNG
   RUNG wire#powerrail
      Contact( "TESTE_LAMPADAS" )
   END_RUNG wire#w1
   RUNG wire#powerrail
      Contact( "Clock_1Hz" )
      Contact( "Multiplo_Uso_DB".EMERGENCIAS_OK )
      wire#w2
      Contact( "DB_Global_Sistema".Apoio_OP10 )
      wire#w3
      Coil( "15MS02_Torre de Sinalização¶Amarela" )
   END_RUNG
   RUNG wire#w2
      Contact( "DB_Global_Sistema".Apoio_OP20 )
   END_RUNG wire#w3
   RUNG wire#w2
      Contact( "DB_Global_Sistema".Apoio_OP30 )
   END_RUNG wire#w3
   RUNG wire#w2
      Contact( "DB_Global_Sistema".Apoio_OP40 )
   END_RUNG wire#w3
   RUNG wire#w2
      Contact( "DB_Global_Sistema".Apoio_OP50 )
   END_RUNG wire#w3
   RUNG wire#w2
      Contact( "DB_Global_Sistema".Apoio_OP60 )
   END_RUNG wire#w3
   RUNG wire#w2
      Contact( "DB_Global_Sistema".Apoio_OP70 )
   END_RUNG wire#w3
   RUNG wire#w2
      Contact( "DB_Global_Sistema".Apoio_OP80 )
   END_RUNG wire#w3
   RUNG wire#w2
      I_Contact( "Multiplo_Uso_DB".EM_JORNADA )
   END_RUNG wire#w3
   RUNG wire#powerrail
      Contact( "TESTE_LAMPADAS" )
   END_RUNG wire#w3
   RUNG wire#powerrail
      Contact( "Clock_1Hz" )
      I_Contact( "Multiplo_Uso_DB".EMERGENCIAS_OK )
      wire#w4
      Coil( "15MS02_Torre de Sinalização¶Vermelha" )
   END_RUNG
   RUNG wire#powerrail
      Contact( "TESTE_LAMPADAS" )
   END_RUNG wire#w4
   // the same network as SCL:
   "15MS02_Torre de Sinalização¶Verde" := ("Multiplo_Uso_DB".EM_JORNADA AND "Multiplo_Uso_DB".IHM_Modo_Automatico AND "Multiplo_Uso_DB".EMERGENCIAS_OK AND NOT "DB_Global_Sistema".Apoio_OP10 AND NOT "DB_Global_Sistema".Apoio_OP20 AND NOT "DB_Global_Sistema".Apoio_OP30 AND NOT "DB_Global_Sistema".Apoio_OP40 AND NOT "DB_Global_Sistema".Apoio_OP50 AND NOT "DB_Global_Sistema".Apoio_OP60 AND NOT "DB_Global_Sistema".Apoio_OP70 AND NOT "DB_Global_Sistema".Apoio_OP80) OR "TESTE_LAMPADAS";
   "15MS02_Torre de Sinalização¶Amarela" := ("Clock_1Hz" AND "Multiplo_Uso_DB".EMERGENCIAS_OK AND ("DB_Global_Sistema".Apoio_OP10 OR "DB_Global_Sistema".Apoio_OP20 OR "DB_Global_Sistema".Apoio_OP30 OR "DB_Global_Sistema".Apoio_OP40 OR "DB_Global_Sistema".Apoio_OP50 OR "DB_Global_Sistema".Apoio_OP60 OR "DB_Global_Sistema".Apoio_OP70 OR "DB_Global_Sistema".Apoio_OP80 OR NOT "Multiplo_Uso_DB".EM_JORNADA)) OR "TESTE_LAMPADAS";
   "15MS02_Torre de Sinalização¶Vermelha" := ("Clock_1Hz" AND NOT "Multiplo_Uso_DB".EMERGENCIAS_OK) OR "TESTE_LAMPADAS";
END_REGION
END_ORGANIZATION_BLOCK

ORGANIZATION_BLOCK "Parada_Operacoes"   // OB124, LAD, ProgramCycle
TITLE = "Main Program Sweep (Cycle)"
{ S7_Optimized_Access := 'TRUE' }
VERSION : 0.1
   VAR_INPUT
      Initial_Call : Bool;   // Initial call of this OB
      Remanence : Bool;   // =True, if remanent data are available
   END_VAR
BEGIN

REGION Network 1: Para OP10
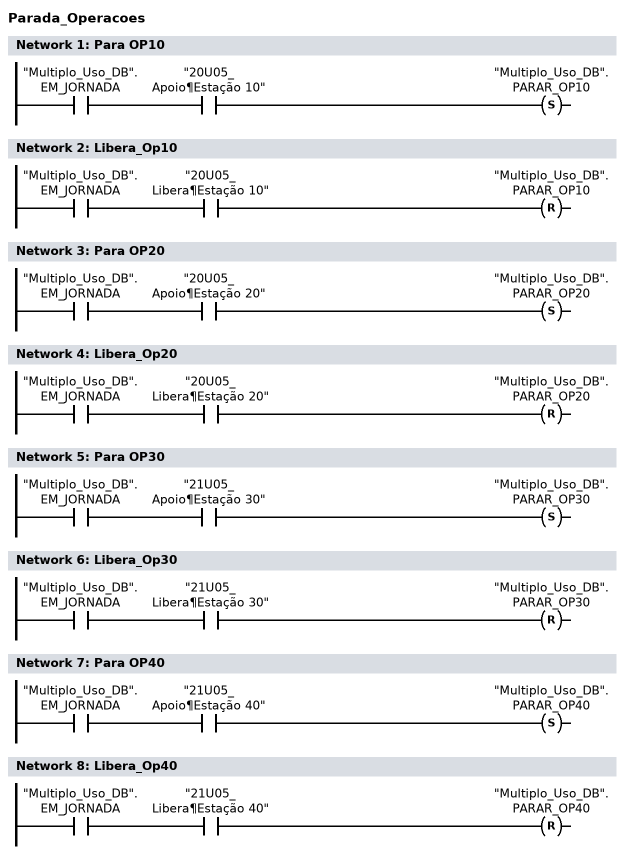
   RUNG wire#powerrail
      Contact( "Multiplo_Uso_DB".EM_JORNADA )
      Contact( "20U05_Apoio¶Estação 10" )
      S_Coil( "Multiplo_Uso_DB".PARAR_OP10 )
   END_RUNG
   // the same network as SCL:
   IF "Multiplo_Uso_DB".EM_JORNADA AND "20U05_Apoio¶Estação 10" THEN
       "Multiplo_Uso_DB".PARAR_OP10 := TRUE;
   END_IF;
END_REGION

REGION Network 2: Libera_Op10
   RUNG wire#powerrail
      Contact( "Multiplo_Uso_DB".EM_JORNADA )
      Contact( "20U05_Libera¶Estação 10" )
      R_Coil( "Multiplo_Uso_DB".PARAR_OP10 )
   END_RUNG
   // the same network as SCL:
   IF "Multiplo_Uso_DB".EM_JORNADA AND "20U05_Libera¶Estação 10" THEN
       "Multiplo_Uso_DB".PARAR_OP10 := FALSE;
   END_IF;
END_REGION

REGION Network 3: Para OP20
   RUNG wire#powerrail
      Contact( "Multiplo_Uso_DB".EM_JORNADA )
      Contact( "20U05_Apoio¶Estação 20" )
      S_Coil( "Multiplo_Uso_DB".PARAR_OP20 )
   END_RUNG
   // the same network as SCL:
   IF "Multiplo_Uso_DB".EM_JORNADA AND "20U05_Apoio¶Estação 20" THEN
       "Multiplo_Uso_DB".PARAR_OP20 := TRUE;
   END_IF;
END_REGION

REGION Network 4: Libera_Op20
   RUNG wire#powerrail
      Contact( "Multiplo_Uso_DB".EM_JORNADA )
      Contact( "20U05_Libera¶Estação 20" )
      R_Coil( "Multiplo_Uso_DB".PARAR_OP20 )
   END_RUNG
   // the same network as SCL:
   IF "Multiplo_Uso_DB".EM_JORNADA AND "20U05_Libera¶Estação 20" THEN
       "Multiplo_Uso_DB".PARAR_OP20 := FALSE;
   END_IF;
END_REGION

REGION Network 5: Para OP30
   RUNG wire#powerrail
      Contact( "Multiplo_Uso_DB".EM_JORNADA )
      Contact( "21U05_Apoio¶Estação 30" )
      S_Coil( "Multiplo_Uso_DB".PARAR_OP30 )
   END_RUNG
   // the same network as SCL:
   IF "Multiplo_Uso_DB".EM_JORNADA AND "21U05_Apoio¶Estação 30" THEN
       "Multiplo_Uso_DB".PARAR_OP30 := TRUE;
   END_IF;
END_REGION

REGION Network 6: Libera_Op30
   RUNG wire#powerrail
      Contact( "Multiplo_Uso_DB".EM_JORNADA )
      Contact( "21U05_Libera¶Estação 30" )
      R_Coil( "Multiplo_Uso_DB".PARAR_OP30 )
   END_RUNG
   // the same network as SCL:
   IF "Multiplo_Uso_DB".EM_JORNADA AND "21U05_Libera¶Estação 30" THEN
       "Multiplo_Uso_DB".PARAR_OP30 := FALSE;
   END_IF;
END_REGION

REGION Network 7: Para OP40
   RUNG wire#powerrail
      Contact( "Multiplo_Uso_DB".EM_JORNADA )
      Contact( "21U05_Apoio¶Estação 40" )
      S_Coil( "Multiplo_Uso_DB".PARAR_OP40 )
   END_RUNG
   // the same network as SCL:
   IF "Multiplo_Uso_DB".EM_JORNADA AND "21U05_Apoio¶Estação 40" THEN
       "Multiplo_Uso_DB".PARAR_OP40 := TRUE;
   END_IF;
END_REGION

REGION Network 8: Libera_Op40
   RUNG wire#powerrail
      Contact( "Multiplo_Uso_DB".EM_JORNADA )
      Contact( "21U05_Libera¶Estação 40" )
      R_Coil( "Multiplo_Uso_DB".PARAR_OP40 )
   END_RUNG
   // the same network as SCL:
   IF "Multiplo_Uso_DB".EM_JORNADA AND "21U05_Libera¶Estação 40" THEN
       "Multiplo_Uso_DB".PARAR_OP40 := FALSE;
   END_IF;
END_REGION
END_ORGANIZATION_BLOCK

(* ===== HMI "HMI_RT_1" =====
system functions are stored by id; their names below are inferred from use
connection "HMI_Connection_1": ETHERNET, S7_1500_OMS

HMI tags "Default tag table"
   "IHM_TESTE" : Int AT %DB1.DBW0
   "Multiplo_Uso_DB_IHM_TAKT_MINUTOS" : Int = PLC Multiplo_Uso_DB.IHM_TAKT_MINUTOS, 1 s
   "Multiplo_Uso_DB_IHM_TAKT_SEGUNDOS" : Int = PLC Multiplo_Uso_DB.IHM_TAKT_SEGUNDOS, 1 s
   "Multiplo_Uso_DB_TAKT_SEGUNDOS" : Int = PLC Multiplo_Uso_DB.TAKT_SEGUNDOS, 1 s
   "Multiplo_Uso_DB_INICIO_JORNADA" : DTL = PLC Multiplo_Uso_DB.INICIO_JORNADA, 1 s
   "Multiplo_Uso_DB_INICIO_ALMOÇO" : DTL = PLC Multiplo_Uso_DB.INICIO_ALMOÇO, 1 s
   "Multiplo_Uso_DB_FINAL_JORNADA" : DTL = PLC Multiplo_Uso_DB.FINAL_JORNADA, 1 s
   "Multiplo_Uso_DB_TOTAL_CABINAS_TURNO" : Int = PLC Multiplo_Uso_DB.TOTAL_CABINAS_TURNO, 1 s
   "IHM_Tempo_Takt" : Time = PLC IHM_Tempo_Takt AT %MD4, 1 s
   "Multiplo_Uso_DB_Emergencia_OP10_OK" : Bool = PLC Multiplo_Uso_DB.Emergencia_OP10_OK, 1 s
   "Multiplo_Uso_DB_Emergencia_OP20_OK" : Bool = PLC Multiplo_Uso_DB.Emergencia_OP20_OK, 1 s
   "Multiplo_Uso_DB_Emergencia_OP30_OK" : Bool = PLC Multiplo_Uso_DB.Emergencia_OP30_OK, 1 s
   "ALARMES_DB_DBW0" : Int = PLC ALARMES_DB.DBW0 AT %DB12.DBW0, 1 s
   "ALARMES_DB_DBW1" : Int = PLC ALARMES_DB.DBW1 AT %DB12.DBW2, 1 s
   "Multiplo_Uso_DB_IHM_Velocidade_Automatico" : Int = PLC Multiplo_Uso_DB.IHM_Velocidade_Automatico, 1 s
   "Multiplo_Uso_DB_IHM_Velocidade_Manual" : Int = PLC Multiplo_Uso_DB.IHM_Velocidade_Manual, 1 s
   "Multiplo_Uso_DB_IHM_Descolamento_Cabinas_mm" : DInt = PLC Multiplo_Uso_DB.IHM_Descolamento_Cabinas_mm, 1 s
   "Multiplo_Uso_DB_IHM_Jog_CCW" : Bool = PLC Multiplo_Uso_DB.IHM_Jog_CCW, 1 s
   "Multiplo_Uso_DB_IHM_Jog_CW" : Bool = PLC Multiplo_Uso_DB.IHM_Jog_CW, 1 s
   "Multiplo_Uso_DB_IHM_Modo_Manual" : Bool = PLC Multiplo_Uso_DB.IHM_Modo_Manual, 1 s
   "Multiplo_Uso_DB_IHM_HABILITA_DRIVER" : Bool = PLC Multiplo_Uso_DB.IHM_HABILITA_DRIVER, 1 s
   "Multiplo_Uso_DB_Emergencia_OP40_OK" : Bool = PLC Multiplo_Uso_DB.Emergencia_OP40_OK, 1 s
   "Multiplo_Uso_DB_Emergencia_OP50_OK" : Bool = PLC Multiplo_Uso_DB.Emergencia_OP50_OK, 1 s
   "Multiplo_Uso_DB_Emergencia_OP60_OK" : Bool = PLC Multiplo_Uso_DB.Emergencia_OP60_OK, 1 s
   "Multiplo_Uso_DB_Emergencia_OP70_OK" : Bool = PLC Multiplo_Uso_DB.Emergencia_OP70_OK, 1 s
   "Multiplo_Uso_DB_Emergencia_OP80_OK" : Bool = PLC Multiplo_Uso_DB.Emergencia_OP80_OK, 1 s
   "Multiplo_Uso_DB_Emergencia_Principal_OK" : Bool = PLC Multiplo_Uso_DB.Emergencia_Principal_OK, 1 s
   "DB_Global_Sistema_TEMPO_TAKT" : Int = PLC DB_Global_Sistema.TEMPO_TAKT AT %DB23.DBW0, 1 s
   "DB_Global_Sistema_Apoio_OP10" : Bool = PLC DB_Global_Sistema.Apoio_OP10 AT %DB23.DBX2.0, 1 s
   "DB_Global_Sistema_Apoio_OP20" : Bool = PLC DB_Global_Sistema.Apoio_OP20 AT %DB23.DBX2.1, 1 s
   "DB_Global_Sistema_Apoio_OP30" : Bool = PLC DB_Global_Sistema.Apoio_OP30 AT %DB23.DBX2.2, 1 s
   "DB_Global_Sistema_Apoio_OP40" : Bool = PLC DB_Global_Sistema.Apoio_OP40 AT %DB23.DBX2.3, 1 s
   "DB_Global_Sistema_Apoio_OP50" : Bool = PLC DB_Global_Sistema.Apoio_OP50 AT %DB23.DBX2.4, 1 s
   "DB_Global_Sistema_Apoio_OP60" : Bool = PLC DB_Global_Sistema.Apoio_OP60 AT %DB23.DBX2.5, 1 s
   "DB_Global_Sistema_Apoio_OP70" : Bool = PLC DB_Global_Sistema.Apoio_OP70 AT %DB23.DBX2.6, 1 s
   "DB_Global_Sistema_Apoio_OP80" : Bool = PLC DB_Global_Sistema.Apoio_OP80 AT %DB23.DBX2.7, 1 s
   "Multiplo_Uso_DB_IHM_Tempo_Aviso2" : Int = PLC Multiplo_Uso_DB.IHM_Tempo_Aviso2, 1 s
   "Multiplo_Uso_DB_IHM_Tempo_Aviso1" : Int = PLC Multiplo_Uso_DB.IHM_Tempo_Aviso1, 1 s
   "23U05_Cabine_Retirada" : Bool = PLC 21U05_Cabine_Retirada AT %I144.4, 1 s
   "Multiplo_Uso_DB_CONTAGEM_CABINAS" : Int = PLC Multiplo_Uso_DB.CONTAGEM_CABINAS, 1 s
   "Multiplo_Uso_DB_IHM_Zerar_Contagem" : Bool = PLC Multiplo_Uso_DB.IHM_Zerar_Contagem, 1 s
   "Multiplo_Uso_DB_IHM_Zerar_Posicao_Esteira" : Bool = PLC Multiplo_Uso_DB.IHM_Zerar_Posicao_Esteira, 1 s
   "Multiplo_Uso_DB_IHM_Posicao_Atual" : DInt = PLC Multiplo_Uso_DB.IHM_Posicao_Atual, 1 s
   "Multiplo_Uso_DB_IHM_Zerar_Takt" : Bool = PLC Multiplo_Uso_DB.IHM_Zerar_Takt, 1 s
   "Multiplo_Uso_DB_HORA_Atual" : Time_Of_Day = PLC Multiplo_Uso_DB.HORA_Atual, 1 s
   "Multiplo_Uso_DB_DATA_Atual" : DTL = PLC Multiplo_Uso_DB.DATA_Atual, 1 s
   "20U1_GRUPO_OK" : Bool = PLC 20U1_GRUPO_OK AT %I25.1, 1 s
   "21U1_GRUPO_OK" : Bool = PLC 21U1_GRUPO_OK AT %I34.1, 1 s
   "TESTE_LAMPADAS" : Bool = PLC TESTE_LAMPADAS AT %M20.0, 1 s

discrete alarms
   1: 'Verificar botão de emergencia da OPeração 10 / FALHA EMERGENCIA PRINCIPAL', class Warnings, trigger "ALARMES_DB_DBW0" bit 0
   2: 'FALHA EMERGENCIA OPERAÇÃO 10', class Warnings, trigger "ALARMES_DB_DBW0" bit 1
   3: 'FALHA EMERGENCIA OPERAÇÃO 20', class Warnings, trigger "ALARMES_DB_DBW0" bit 2
   4: 'FALHA EMERGENCIA OPERAÇÃO 30', class Warnings, trigger "ALARMES_DB_DBW0" bit 3
   5: 'FALHA EMERGENCIA OPERAÇÃO 40', class Warnings, trigger "ALARMES_DB_DBW0" bit 4
   6: 'FALHA EMERGENCIA OPERAÇÃO 50', class Warnings, trigger "ALARMES_DB_DBW0" bit 5
   7: 'FALHA EMERGENCIA OPERAÇÃO 60', class Warnings, trigger "ALARMES_DB_DBW0" bit 6
   8: 'FALHA EMERGENCIA OPERAÇÃO 70', class Warnings, trigger "ALARMES_DB_DBW0" bit 7
   9: 'FALHA EMERGENCIA OPERAÇÃO 80', class Warnings, trigger "ALARMES_DB_DBW0" bit 8
   10: 'VERIFICAR TEMPERATURA DO PAINEL', class MIKROMAQ, trigger "ALARMES_DB_DBW0" bit 9
   11: 'VERIFICAR DISJUNTOR DE SERVIÇO 07F00', class MIKROMAQ, trigger "ALARMES_DB_DBW0" bit 10
   12: 'VERIFICAR DISJUNTOR TOMADAS 07F03', class MIKROMAQ, trigger "ALARMES_DB_DBW0" bit 11
   13: 'VERIFICAR DISJUNTOR ILUMINAÇÃO 07F04', class MIKROMAQ, trigger "ALARMES_DB_DBW0" bit 12
   14: 'VERIFICAR DISJUNTOR AR CONDICIONADO 07F06', class MIKROMAQ, trigger "ALARMES_DB_DBW0" bit 13
   15: 'FALHA NO DISJUNTOR 08F03', class Warnings, trigger "ALARMES_DB_DBW0" bit 14
   16: 'FALHA NO DISJUNTOR FREIO 09F01', class Warnings, trigger "ALARMES_DB_DBW0" bit 15
   18: 'SOBREAQUECIMENO RESISTOR FRENAGEM 09F04', class Warnings, trigger "ALARMES_DB_DBW1" bit 1
   19: 'FALHA NO DISJUNTOR DA VENTILAÇÃO DO DRIVER 09F06', class Warnings, trigger "ALARMES_DB_DBW1" bit 2
   20: 'CORTINA DE SAIDA ACIONADA DURANTE GIRO', class Warnings, trigger "ALARMES_DB_DBW1" bit 3
   17: 'FALHA NO INVERSOR', class Warnings, trigger "ALARMES_DB_DBW1" bit 0

graphic list "Graphic_list_1": 0 'emergencia'; 1 'painel'

Template "Comum" 800x480
   GraphicView "Template_Graphic view_1" at 1,0 size 205x75; Picture "LogoScania"
   DateTimeField "Template_Date/time field_1" at 635,7 size 123x26
   DateTimeField "Template_Date/time field_2" at 637,43 size 126x26

screen "Main" 800x480, template "Comum"
   TextField "Text field_1" at 343,10 size 111x47; Text 'MAIN'
   Button "Button_1" at 8,440 size 164x37; TextOff 'PRODUÇÃO'; Authorization "Monitor"
      on Release: ActivateScreen("PRODUCAO", 0)
   Button "Button_2" at 214,440 size 164x37; TextOff 'MANUTENÇÃO'; Authorization "Operate"
      on Release: ActivateScreen("MANUTENCAO", 0)
   Button "Button_3" at 421,440 size 164x37; TextOff 'ENGENHARIA'; Authorization "User administration"
      on Release: ActivateScreen("ENGENHARIA", 0)
   Button "Button_4" at 628,440 size 164x37; TextOff 'LOGIN'
      on Release: function_a2a04561()
   GraphicView "Graphic view_1" at 2,80 size 796x356; Picture "TOPOLOGIA_LINHA03"
   GraphicView "Graphic view_2" at 131,319 size 34x24; Picture "emergencia"
      Appearance <- "Multiplo_Uso_DB_Emergencia_OP10_OK"
      Visibility <- "Multiplo_Uso_DB_Emergencia_OP10_OK"
   GraphicView "Graphic view_3" at 173,319 size 34x24; Picture "emergencia"
      Appearance <- "Multiplo_Uso_DB_Emergencia_OP20_OK"
      Visibility <- "Multiplo_Uso_DB_Emergencia_OP20_OK"
   GraphicView "Graphic view_4" at 400,319 size 34x24; Picture "emergencia"
      Appearance <- "Multiplo_Uso_DB_Emergencia_OP30_OK"
      Visibility <- "Multiplo_Uso_DB_Emergencia_OP30_OK"
   GraphicView "Graphic view_5" at 441,320 size 34x24; Picture "emergencia"
      Appearance <- "Multiplo_Uso_DB_Emergencia_OP40_OK"
      Visibility <- "Multiplo_Uso_DB_Emergencia_OP40_OK"
   GraphicView "Graphic view_10" at 629,126 size 34x24; Picture "emergencia"
      Appearance <- "Multiplo_Uso_DB_Emergencia_Principal_OK"
      Visibility <- "Multiplo_Uso_DB_Emergencia_Principal_OK"
   GraphicView "Graphic view_6" at 162,261 size 21x38; Picture "X"
      Appearance <- "20U1_GRUPO_OK"
      Visibility <- "20U1_GRUPO_OK"
   GraphicView "Graphic view_11" at 426,261 size 21x38; Picture "X"
      Appearance <- "21U1_GRUPO_OK"
      Visibility <- "21U1_GRUPO_OK"

screen "ENGENHARIA" 800x480, template "Comum"
   TextField "Text field_1" at 271,12 size 263x47; Text 'ENGENHARIA'
   TextField "Text field_3" at 30,93 size 306x28; Text 'VELOCIDADE DE PROCESSO'
   TextField "Text field_4" at 30,134 size 232x28; Text 'VELOCIDADE DE JOG'
   TextField "Text field_5" at 30,175 size 242x28; Text 'AVANÇO POR CABINA'
   Button "FB_Plus_Rectangular" at 165,327 size 134x50; TextOff 'Text'; PictureOff "FB_Plus_Rectangular_Released_256c"; PictureOn "FB_Plus_Rectangular_Pressed_256c"
      on Press: SetBit("Multiplo_Uso_DB_IHM_Jog_CW")
      on Release: ResetBit("Multiplo_Uso_DB_IHM_Jog_CW")
   Button "FB_Minus_Rectangular" at 23,327 size 134x50; TextOff 'Text'; PictureOff "FB_Minus_Rectangular_Released_256c"; PictureOn "FB_Minus_Rectangular_Pressed_256c"
      on Press: SetBit("Multiplo_Uso_DB_IHM_Jog_CCW")
      on Release: ResetBit("Multiplo_Uso_DB_IHM_Jog_CCW")
   Switch "Toggle_Horizontal_GN" at 491,298 size 276x42; TextOn 'MANUAL / 1'; TextOff 'AUTO / 0'; CaptionText 'Switch'; PictureOff "Toggle_Horizontal_GN_Off_256c"; PictureOn "Toggle_Horizontal_GN_On_256c"
      ProcessValue <- "Multiplo_Uso_DB_IHM_Modo_Manual"
   Switch "Toggle_Horizontal_GN_1" at 492,375 size 276x42; TextOn 'DRIVER ON / 1'; TextOff 'DRIVER OFF / 0'; CaptionText 'Switch'; PictureOff "Toggle_Horizontal_GN_Off_256c"; PictureOn "Toggle_Horizontal_GN_On_256c"
      ProcessValue <- "Multiplo_Uso_DB_IHM_HABILITA_DRIVER"
   TextField "Text field_6" at 495,264 size 283x34; Text 'DRIVE AUTO / MANU'
   TextField "Text field_7" at 519,343 size 230x34; Text 'HABILITA DRIVE'
   TextField "Text field_8" at 58,269 size 206x34; Text 'COMANDO JOG'
   Button "SB_ExitRuntime_85x64" at 353,352 size 85x64; TextOff 'Text'; PictureOff "SB_ExitRuntime_85x64_256c"
      on Click: StopRuntime(0)
   TextField "Text field_9" at 360,312 size 72x34; Text 'SAIR'
   TextField "Text field_10" at 365,272 size 61x34; Text 'IHM'
   Button "Button_1" at 8,440 size 164x37; TextOff 'MAIN'; Authorization "User administration"
      on Change: ActivateScreen("Main", 0)
   Button "Button_4" at 627,439 size 164x37; TextOff 'ALARMES'; TextOn 'STATUS CLP'
      on Release: ActivateScreen("ALARMES", 0)
   TextField "Text field_2" at 30,216 size 285x28; Text 'POSIÇÃO ATUAL ESTEIRA'
   IOField "I/O field_1" at 346,91 size 96x32; FormatPattern 99; Unit mm/s
      ProcessValue <- "Multiplo_Uso_DB_IHM_Velocidade_Automatico"
   IOField "I/O field_2" at 346,132 size 96x32; FormatPattern 99; Unit mm/s
      ProcessValue <- "Multiplo_Uso_DB_IHM_Velocidade_Manual"
   IOField "I/O field_3" at 346,173 size 96x32; FormatPattern 9999; Unit mm
      ProcessValue <- "Multiplo_Uso_DB_IHM_Descolamento_Cabinas_mm"
   IOField "I/O field_4" at 346,214 size 96x32; FormatPattern 99999; Unit mm
      ProcessValue <- "Multiplo_Uso_DB_IHM_Posicao_Atual"
   Button "Button_2" at 490,183 size 280x42; TextOff 'ZERAR POSIÇÃO'
      on Press: SetBit("Multiplo_Uso_DB_IHM_Zerar_Posicao_Esteira")
      on Release: ResetBit("Multiplo_Uso_DB_IHM_Zerar_Posicao_Esteira")
   TextField "Text field_11" at 522,93 size 225x34; Text 'ZERAR POSIÇÃO'
   TextField "Text field_12" at 575,125 size 120x34; Text 'ESTEIRA'

screen "PRODUCAO" 800x480, template "Comum"
   TextField "Text field_1" at 292,12 size 222x47; Text 'PRODUÇÃO'
   Button "Button_1" at 8,441 size 164x37; TextOff 'MAIN'; Authorization "Monitor"
      on Change: ActivateScreen("Main", 0)
   Button "Button_2" at 214,441 size 164x37; TextOff 'TAKT TIME'; Authorization "Monitor"
      on Release: ActivateScreen("TAKT TIME", 0)
   Button "Button_3" at 420,441 size 164x37; TextOff 'ANDON'; Authorization "Monitor"
      on Release: ActivateScreen("ANDON", 0)
   Button "Button_4" at 627,440 size 164x37; TextOff 'ALARMES'; TextOn 'STATUS CLP'
      on Release: ActivateScreen("ALARMES", 0)
   GraphicView "Graphic view_1" at 2,80 size 796x356; Picture "TOPOLOGIA_LINHA03"
   GraphicView "Graphic view_2" at 131,319 size 34x24; Picture "emergencia"
      Appearance <- "Multiplo_Uso_DB_Emergencia_OP10_OK"
      Visibility <- "Multiplo_Uso_DB_Emergencia_OP10_OK"
   GraphicView "Graphic view_3" at 173,319 size 34x24; Picture "emergencia"
      Appearance <- "Multiplo_Uso_DB_Emergencia_OP20_OK"
      Visibility <- "Multiplo_Uso_DB_Emergencia_OP20_OK"
   GraphicView "Graphic view_4" at 400,319 size 34x24; Picture "emergencia"
      Appearance <- "Multiplo_Uso_DB_Emergencia_OP30_OK"
      Visibility <- "Multiplo_Uso_DB_Emergencia_OP30_OK"
   GraphicView "Graphic view_5" at 441,320 size 34x24; Picture "emergencia"
      Appearance <- "Multiplo_Uso_DB_Emergencia_OP40_OK"
      Visibility <- "Multiplo_Uso_DB_Emergencia_OP40_OK"
   GraphicView "Graphic view_10" at 629,126 size 34x24; Picture "emergencia"
      Appearance <- "Multiplo_Uso_DB_Emergencia_Principal_OK"
      Visibility <- "Multiplo_Uso_DB_Emergencia_Principal_OK"
   GraphicView "Graphic view_6" at 162,261 size 21x38; Picture "X"
      Appearance <- "20U1_GRUPO_OK"
      Visibility <- "20U1_GRUPO_OK"
   GraphicView "Graphic view_11" at 426,261 size 21x38; Picture "X"
      Appearance <- "21U1_GRUPO_OK"
      Visibility <- "21U1_GRUPO_OK"

screen "MANUTENCAO" 800x480, template "Comum"
   TextField "Text field_1" at 265,12 size 276x47; Text 'MANUTENÇÃO'
   Button "Button_2" at 168,441 size 142x37; TextOff 'EMERGENCIA'; TextOn 'STATUS EMERGENCIA'; Authorization "Operate"
      on Release: ActivateScreen("EMERGENCIA", 0)
   Button "Button_3" at 329,441 size 142x37; TextOff 'REDE'; TextOn 'STATUS REDE'; Authorization "Operate"
      on Release: ActivateScreen("REDE", 0)
   Button "Button_4" at 651,440 size 142x37; TextOff 'ALARMES'; TextOn 'STATUS CLP'
      on Release: ActivateScreen("ALARMES", 0)
   Button "Button_6" at 8,441 size 142x37; TextOff 'MAIN'; Authorization "Operate"
      on Change: ActivateScreen("Main", 0)
   GraphicView "Graphic view_1" at 2,80 size 796x356; Picture "TOPOLOGIA_LINHA03"
   GraphicView "Graphic view_2" at 131,319 size 34x24; Picture "emergencia"
      Appearance <- "Multiplo_Uso_DB_Emergencia_OP10_OK"
      Visibility <- "Multiplo_Uso_DB_Emergencia_OP10_OK"
   GraphicView "Graphic view_3" at 173,319 size 34x24; Picture "emergencia"
      Appearance <- "Multiplo_Uso_DB_Emergencia_OP20_OK"
      Visibility <- "Multiplo_Uso_DB_Emergencia_OP20_OK"
   GraphicView "Graphic view_4" at 400,319 size 34x24; Picture "emergencia"
      Appearance <- "Multiplo_Uso_DB_Emergencia_OP30_OK"
      Visibility <- "Multiplo_Uso_DB_Emergencia_OP30_OK"
   GraphicView "Graphic view_5" at 441,320 size 34x24; Picture "emergencia"
      Appearance <- "Multiplo_Uso_DB_Emergencia_OP40_OK"
      Visibility <- "Multiplo_Uso_DB_Emergencia_OP40_OK"
   GraphicView "Graphic view_10" at 629,126 size 34x24; Picture "emergencia"
      Appearance <- "Multiplo_Uso_DB_Emergencia_Principal_OK"
      Visibility <- "Multiplo_Uso_DB_Emergencia_Principal_OK"
   GraphicView "Graphic view_6" at 162,261 size 21x38; Picture "X"
      Appearance <- "20U1_GRUPO_OK"
      Visibility <- "20U1_GRUPO_OK"
   GraphicView "Graphic view_11" at 426,261 size 21x38; Picture "X"
      Appearance <- "21U1_GRUPO_OK"
      Visibility <- "21U1_GRUPO_OK"
   Button "Button_1" at 490,440 size 142x37; TextOn 'STATUS REDE'; TextOff 'TESTE LAMP'; Authorization "Operate"
      on Press: SetBit("TESTE_LAMPADAS")
      on Release: ResetBit("TESTE_LAMPADAS")

screen "EMERGENCIA OLD" 800x480, template "Comum"
   GraphicView "Graphic view_1" at 10,82 size 780x326; Picture "ESTACOES8_1"
   TextField "Text field_1" at 49,241 size 47x20; Text 'OP.10'
   TextField "Text field_2" at 130,241 size 47x20; Text 'OP.20'
   TextField "Text field_3" at 226,241 size 47x20; Text 'OP.30'
   TextField "Text field_4" at 322,241 size 47x20; Text 'OP.40'
   TextField "Text field_5" at 421,241 size 47x20; Text 'OP.50'
   TextField "Text field_6" at 524,241 size 47x20; Text 'OP.60'
   TextField "Text field_7" at 624,241 size 47x20; Text 'OP.70'
   TextField "Text field_8" at 715,241 size 47x20; Text 'OP.80'
   Group "Group" at 10,82 size 780x326; Picture "ESTACOES8_1"
   TextField "Text field_9" at 271,12 size 260x47; Text 'EMERGÊNCIA'
   GraphicView "Graphic view_2" at 50,313 size 30x30; Picture "emergencia"
      Appearance <- "Multiplo_Uso_DB_Emergencia_OP10_OK"
   GraphicView "Graphic view_3" at 134,313 size 30x30; Picture "emergencia"
      Appearance <- "Multiplo_Uso_DB_Emergencia_OP20_OK"
   GraphicView "Graphic view_4" at 234,313 size 30x30; Picture "emergencia"
      Appearance <- "Multiplo_Uso_DB_Emergencia_OP30_OK"
   GraphicView "Graphic view_5" at 329,313 size 30x30; Picture "emergencia"
      Appearance <- "Multiplo_Uso_DB_Emergencia_OP40_OK"
   Button "Button_1" at 677,412 size 121x68; TextOff 'VOLTAR'
      on Press: ActivateScreen("MANUTENCAO", 0)
   GraphicView "Graphic view_10" at 680,100 size 50x40; Picture "emergencia"
      Appearance <- "Multiplo_Uso_DB_Emergencia_Principal_OK"
   TextField "Text field_10" at 650,140 size 117x20; Text 'Painel Principal'

screen "REDE" 800x480, template "Comum"
   TextField "Text field_9" at 283,10 size 271x47; Text 'ESTADO REDE'
   TextField "Text field_6" at 26,198 size 152x20; Text 'ELEVADOR ENTRADA'
   GraphicView "Graphic view_9" at 72,104 size 99x88; Picture "MURR U05"
   TextField "Text field_12" at 97,102 size 50x20; Text '20U01'
   TextField "Text field_13" at 97,144 size 50x20; Text '20U05'
   GraphicView "Graphic view_13" at 383,322 size 42x61; Picture "19U02"
   TextField "Text field_20" at 381,318 size 50x20; Text '19U02'
   GraphicView "Graphic view_2" at 74,106 size 96x83; Picture "X"
      Appearance <- "20U1_GRUPO_OK"
      Visibility <- "20U1_GRUPO_OK"
   Button "Button_2" at 16,440 size 164x37; TextOff 'VOLTAR'; Authorization "Operate"
      on Change: ActivateScreen("MANUTENCAO", 0)
   Button "Button_4" at 630,440 size 164x37; TextOff 'ALARMES'; TextOn 'STATUS CLP'
      on Release: ActivateScreen("ALARMES", 0)
   GraphicView "Graphic view_1" at 22,204 size 767x92; Picture "LINHA01"
   GraphicView "Graphic view_3" at 63,273 size 37x21; Picture "Right_Arrow"
   GraphicView "Graphic view_4" at 143,273 size 37x21; Picture "Right_Arrow"
   GraphicView "Graphic view_5" at 239,273 size 37x21; Picture "Right_Arrow"
   GraphicView "Graphic view_6" at 332,273 size 37x21; Picture "Right_Arrow"
   GraphicView "Graphic view_7" at 431,273 size 37x21; Picture "Right_Arrow"
   GraphicView "Graphic view_17" at 534,273 size 37x21; Picture "Right_Arrow"
   GraphicView "Graphic view_18" at 628,273 size 37x21; Picture "Right_Arrow"
   GraphicView "Graphic view_19" at 717,273 size 37x21; Picture "Right_Arrow"
   TextField "Text field_2" at 60,240 size 47x20; Text 'OP.10'
   TextField "Text field_3" at 140,240 size 47x20; Text 'OP.20'
   TextField "Text field_4" at 236,240 size 47x20; Text 'OP.30'
   TextField "Text field_5" at 329,240 size 47x20; Text 'OP.40'
   TextField "Text field_21" at 428,240 size 47x20; Text 'OP.50'
   TextField "Text field_22" at 530,240 size 47x20; Text 'OP.60'
   TextField "Text field_23" at 624,240 size 47x20; Text 'OP.70'
   TextField "Text field_24" at 712,240 size 47x20; Text 'OP.80'
   GraphicView "Graphic view_8" at 253,104 size 99x88; Picture "MURR U05"
   TextField "Text field_14" at 278,102 size 50x20; Text '21U01'
   TextField "Text field_15" at 278,144 size 50x20; Text '21U05'
   GraphicView "Graphic view_11" at 255,106 size 96x83; Picture "X"
      Appearance <- "21U1_GRUPO_OK"
      Visibility <- "21U1_GRUPO_OK"

